RoboDK station: IRB120 3d print.rdk

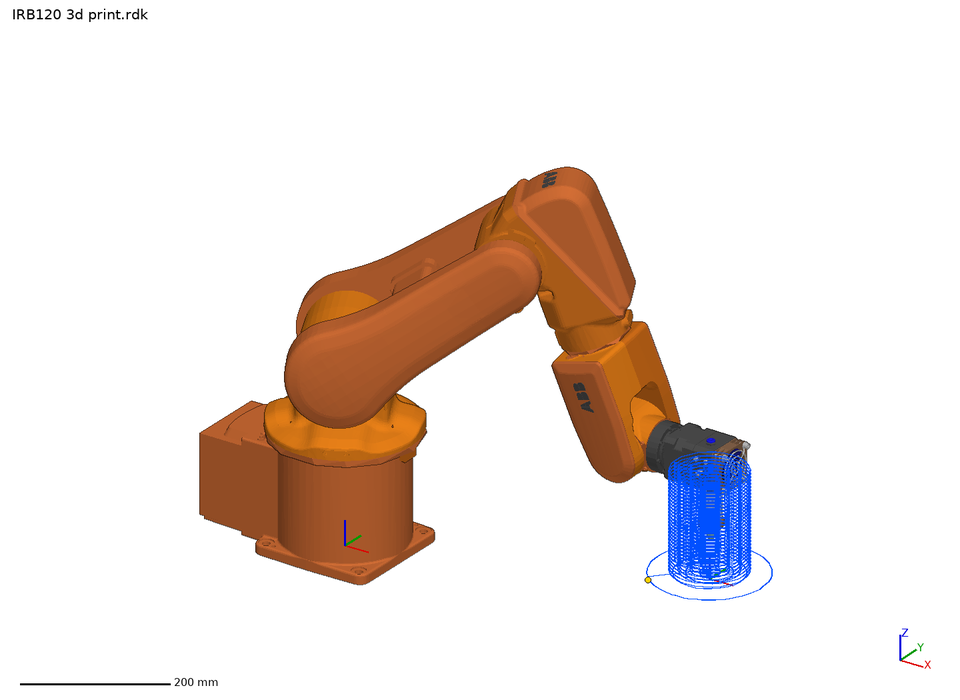
[picture v0: the station drawn from its stored meshes, robots at their saved joint values, targets as dots, program paths as lines]
Station IRB120 3d print (saved by RoboDK 5.2.1). Poses are relative to the parent item; angles as X-Y-Z fixed-axis rotations.
  - frame ABB IRB 120-3/0.6 Base at (0, 0, 0) mm
    - robot ABB IRB 120-3/0.6: 6 axes, payload 3 kg, reach 580 mm, repeatability 0.01 mm, weight 25 kg
        modified DH rows (alpha deg, a mm, theta deg, d mm): 0, 0, 0, 290; -90, 0, -90, 0; 0, 270, 0, 0; -90, 70, 0, 302; 90, 0, 0, 0; -90, 0, 180, 72
        joint limits [-165, -110, -90, -160, -120, -400] to [165, 110, 70, 160, 120, 400]; home [0, 0, 0, 0, 0, 0]; saved at [28.559, 55.09, 16.06, -150.095, 73.514, -189.27]
      - tool Extruder, TCP at (111.33, -10.17, 60.98) mm, rotated rx 0 ry 90 rz 0 deg, size 148.5 x 72.7 x 98.2 mm
  - frame Frame 2 at (454.66, 194.92, 0) mm
    - object Part at (0, 0, 0) mm, size 120 x 120 x 160 mm, geometry from part.sld
  - machining project Print3D settings: C:/Users/Albert/AppData/Local/Temp/Part.stl | rotZ(0) | rotX(0)*rotY(0) | rotZ(0)
  - program Print3D (7572 instructions, listed below)
  - Python program Extruder (listed below)
  - Python program SimulateFinalResult (listed below)
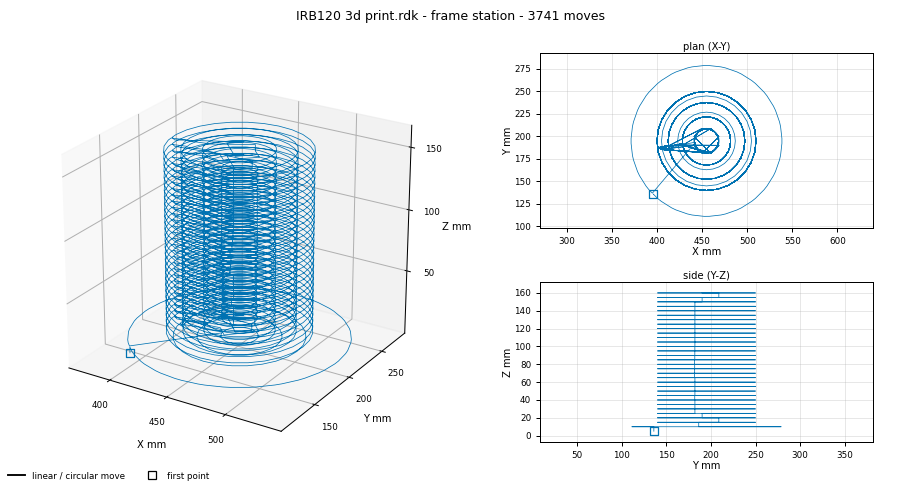
[picture p0: tool path of IRB120 3d print.rdk in frame station, 3741 of 3741 moves have a stored position in this frame; points joined in program order, loops and branches not executed]

--- program Print3D (robot ABB IRB 120-3/0.6) ---
  Set Ref.: Frame 2
  Set Tool: Extruder
  Show Extruder
  Set speed (1000.0 mm/s)
  MoveJ 1 to (-59.03, -59.03, 5) mm, rotated rx 180 ry 0 rz 180 deg; joints [29.08, 61.286, 29.9, -150.915, 91.037, -179.423]
  Set speed (83.3 mm/s)
  MoveL 2 to (-59.03, -59.03, 5) mm, rotated rx 180 ry 0 rz 180 deg; joints [29.08, 61.286, 29.9, -150.915, 91.037, -179.423]
  Call Extruder(-1)
  MoveL 3 to (-59.03, -59.03, 5) mm, rotated rx 180 ry 0 rz 180 deg; joints [29.08, 61.286, 29.9, -150.915, 91.037, -179.423]
  Call Extruder(0.000)
  Set speed (130.0 mm/s)
  MoveL 4 to (-59.03, -59.03, 10) mm, rotated rx 180 ry 0 rz 180 deg; joints [29.08, 60.2, 30.513, -150.918, 90.624, -179.653]
  Call Extruder(-2.000)
  Set speed (40.0 mm/s)
  MoveL 5 to (-59.03, -59.03, 10) mm, rotated rx 180 ry 0 rz 180 deg; joints [29.08, 60.2, 30.513, -150.918, 90.624, -179.653]
  Call Extruder(0.000)
  Set speed (130.0 mm/s)
  MoveL 6 to (-59.03, -59.03, 10) mm, rotated rx 180 ry 0 rz 180 deg; joints [29.08, 60.2, 30.513, -150.918, 90.624, -179.653]
  Call Extruder(2.000)
  Set speed (40.0 mm/s)
  MoveL 7 to (-59.03, -59.03, 10) mm, rotated rx 180 ry 0 rz 180 deg; joints [29.08, 60.2, 30.513, -150.918, 90.624, -179.653]
  Call Extruder(25.861)
  Set speed (30.0 mm/s)
  MoveL 8 to (-54.28, -63.78, 10) mm, rotated rx 180 ry 0 rz 180 deg; joints [27.856, 60.292, 30.1, -152.143, 90.347, -179.817]
  Call Extruder(44.833)
  MoveL 9 to (-50.1, -67.11, 10) mm, rotated rx 180 ry 0 rz -180 deg; joints [26.935, 60.399, 29.628, -153.065, 90.024, -179.988]
  Call Extruder(92.557)
  MoveL 10 to (-38.72, -74.26, 10) mm, rotated rx -180 ry 0 rz -180 deg; joints [24.816, 60.769, 28.068, -155.179, 88.944, -180.488]
  Call Extruder(111.531)
  MoveL 11 to (-33.91, -76.57, 10) mm, rotated rx 180 ry 0 rz 180 deg; joints [24.067, 60.957, 27.309, -155.924, 88.416, -180.708]
  Call Extruder(159.254)
  MoveL 12 to (-21.23, -81.01, 10) mm, rotated rx -180 ry 0 rz -180 deg; joints [22.441, 61.537, 25.081, -157.524, 86.874, -181.292]
  Call Extruder(178.226)
  MoveL 13 to (-16.02, -82.2, 10) mm, rotated rx 180 ry 0 rz 180 deg; joints [21.904, 61.811, 24.081, -158.045, 86.189, -181.535]
  Call Extruder(225.949)
  MoveL 14 to (-2.67, -83.7, 10) mm, rotated rx -180 ry 0 rz -180 deg; joints [20.833, 62.608, 21.313, -159.059, 84.319, -182.169]
  Call Extruder(244.922)
  MoveL 15 to (2.67, -83.7, 10) mm, rotated rx -180 ry 0 rz 180 deg; joints [20.519, 62.966, 20.126, -159.343, 83.532, -182.432]
  Call Extruder(246.414)
  MoveL 16 to (3.09, -83.66, 10) mm, rotated rx 180 ry 0 rz 180 deg; joints [20.502, 62.996, 20.028, -159.358, 83.468, -182.454]
  Call Extruder(292.645)
  MoveL 17 to (16.02, -82.2, 10) mm, rotated rx 180 ry 0 rz 180 deg; joints [19.998, 63.964, 16.96, -159.769, 81.476, -183.127]
  Call Extruder(311.617)
  MoveL 18 to (21.23, -81.01, 10) mm, rotated rx 180 ry 0 rz 180 deg; joints [19.893, 64.397, 15.644, -159.827, 80.641, -183.419]
  Call Extruder(359.340)
  MoveL 19 to (33.91, -76.57, 10) mm, rotated rx -180 ry 0 rz 180 deg; joints [19.872, 65.563, 12.228, -159.706, 78.528, -184.207]
  Call Extruder(378.314)
  MoveL 20 to (38.72, -74.26, 10) mm, rotated rx 180 ry 0 rz -180 deg; joints [19.953, 66.052, 10.842, -159.557, 77.694, -184.542]
  Call Extruder(426.038)
  MoveL 21 to (50.1, -67.11, 10) mm, rotated rx -180 ry 0 rz 180 deg; joints [20.363, 67.333, 7.324, -158.949, 75.638, -185.453]
  Call Extruder(445.010)
  MoveL 22 to (54.28, -63.78, 10) mm, rotated rx -180 ry 0 rz -180 deg; joints [20.601, 67.856, 5.929, -158.621, 74.847, -185.843]
  Call Extruder(492.732)
  MoveL 23 to (63.78, -54.28, 10) mm, rotated rx 180 ry 0 rz -180 deg; joints [21.369, 69.187, 2.461, -157.596, 72.95, -186.892]
  Call Extruder(511.705)
  MoveL 24 to (67.11, -50.1, 10) mm, rotated rx 180 ry 0 rz 180 deg; joints [21.736, 69.715, 1.116, -157.117, 72.241, -187.336]
  Call Extruder(559.428)
  MoveL 25 to (74.26, -38.72, 10) mm, rotated rx -180 ry 0 rz -180 deg; joints [22.792, 71.021, -2.147, -155.749, 70.593, -188.513]
  Call Extruder(578.402)
  MoveL 26 to (76.57, -33.91, 10) mm, rotated rx 180 ry 0 rz -180 deg; joints [23.26, 71.524, -3.38, -155.15, 70, -189.001]
  Call Extruder(626.125)
  MoveL 27 to (81.01, -21.23, 10) mm, rotated rx 180 ry 0 rz 180 deg; joints [24.541, 72.722, -6.277, -153.522, 68.682, -190.264]
  Call Extruder(645.097)
  MoveL 28 to (82.2, -16.02, 10) mm, rotated rx -180 ry 0 rz -180 deg; joints [25.087, 73.164, -7.333, -152.836, 68.235, -190.773]
  Call Extruder(692.820)
  MoveL 29 to (83.7, -2.67, 10) mm, rotated rx 180 ry 0 rz -180 deg; joints [26.535, 74.169, -9.705, -151.04, 67.315, -192.048]
  Call Extruder(711.794)
  MoveL 30 to (83.7, 2.67, 10) mm, rotated rx 180 ry 0 rz -180 deg; joints [27.136, 74.518, -10.521, -150.306, 67.036, -192.543]
  Call Extruder(759.517)
  MoveL 31 to (82.2, 16.02, 10) mm, rotated rx 180 ry 0 rz 180 deg; joints [28.7, 75.248, -12.216, -148.438, 66.561, -193.731]
  Call Extruder(778.488)
  MoveL 32 to (81.01, 21.23, 10) mm, rotated rx 180 ry 0 rz -180 deg; joints [29.338, 75.474, -12.736, -147.696, 66.465, -194.17]
  Call Extruder(826.211)
  MoveL 33 to (76.57, 33.91, 10) mm, rotated rx 180 ry 0 rz -180 deg; joints [30.97, 75.863, -13.631, -145.853, 66.455, -195.16]
  Call Extruder(845.186)
  MoveL 34 to (74.26, 38.72, 10) mm, rotated rx 180 ry 0 rz 180 deg; joints [31.625, 75.944, -13.816, -145.138, 66.542, -195.499]
  Call Extruder(892.909)
  MoveL 35 to (67.11, 50.1, 10) mm, rotated rx 180 ry 0 rz 180 deg; joints [33.281, 75.955, -13.842, -143.401, 66.982, -196.192]
  Call Extruder(911.881)
  MoveL 36 to (63.78, 54.28, 10) mm, rotated rx 180 ry 0 rz 180 deg; joints [33.937, 75.884, -13.678, -142.741, 67.241, -196.398]
  Call Extruder(959.604)
  MoveL 37 to (54.28, 63.78, 10) mm, rotated rx 180 ry 0 rz 180 deg; joints [35.572, 75.515, -12.832, -141.168, 68.083, -196.723]
  Call Extruder(978.576)
  MoveL 38 to (50.1, 67.11, 10) mm, rotated rx 180 ry 0 rz 180 deg; joints [36.21, 75.298, -12.331, -140.581, 68.487, -196.774]
  Call Extruder(1026.299)
  MoveL 39 to (38.72, 74.26, 10) mm, rotated rx -180 ry 0 rz 180 deg; joints [37.78, 74.586, -10.68, -139.203, 69.657, -196.701]
  Call Extruder(1045.274)
  MoveL 40 to (33.91, 76.57, 10) mm, rotated rx -180 ry 0 rz 180 deg; joints [38.384, 74.244, -9.88, -138.697, 70.175, -196.593]
  Call Extruder(1092.996)
  MoveL 41 to (21.23, 81.01, 10) mm, rotated rx 180 ry 0 rz -180 deg; joints [39.84, 73.253, -7.544, -137.529, 71.587, -196.127]
  Call Extruder(1111.968)
  MoveL 42 to (16.02, 82.2, 10) mm, rotated rx 180 ry 0 rz 180 deg; joints [40.39, 72.815, -6.501, -137.108, 72.183, -195.868]
  Call Extruder(1159.691)
  MoveL 43 to (2.67, 83.7, 10) mm, rotated rx 180 ry 0 rz -180 deg; joints [41.682, 71.626, -3.63, -136.158, 73.751, -195.042]
  Call Extruder(1178.665)
  MoveL 44 to (-2.67, 83.7, 10) mm, rotated rx 180 ry 0 rz -180 deg; joints [42.155, 71.126, -2.405, -135.827, 74.393, -194.649]
  Call Extruder(1226.388)
  MoveL 45 to (-16.02, 82.2, 10) mm, rotated rx 180 ry 0 rz -180 deg; joints [43.227, 69.824, 0.84, -135.111, 76.039, -193.513]
  Call Extruder(1245.360)
  MoveL 46 to (-21.23, 81.01, 10) mm, rotated rx 180 ry 0 rz -180 deg; joints [43.6, 69.297, 2.181, -134.877, 76.7, -193.009]
  Call Extruder(1293.082)
  MoveL 47 to (-33.91, 76.57, 10) mm, rotated rx -180 ry 0 rz -180 deg; joints [44.387, 67.965, 5.64, -134.424, 78.363, -191.629]
  Call Extruder(1312.057)
  MoveL 48 to (-38.72, 74.26, 10) mm, rotated rx 180 ry 0 rz -180 deg; joints [44.633, 67.441, 7.035, -134.302, 79.021, -191.043]
  Call Extruder(1359.780)
  MoveL 49 to (-50.1, 67.11, 10) mm, rotated rx 180 ry 0 rz 180 deg; joints [45.066, 66.155, 10.554, -134.156, 80.655, -189.494]
  Call Extruder(1378.752)
  MoveL 50 to (-54.28, 63.78, 10) mm, rotated rx -180 ry 0 rz -180 deg; joints [45.158, 65.663, 11.942, -134.167, 81.294, -188.857]
  Call Extruder(1380.244)
  MoveL 51 to (-54.57, 63.48, 10) mm, rotated rx 180 ry 0 rz 180 deg; joints [45.158, 65.625, 12.051, -134.174, 81.343, -188.806]
  Call Extruder(1426.475)
  MoveL 52 to (-63.78, 54.28, 10) mm, rotated rx 180 ry 0 rz 180 deg; joints [45.163, 64.489, 15.368, -134.385, 82.867, -187.23]
  Call Extruder(1445.447)
  MoveL 53 to (-67.11, 50.1, 10) mm, rotated rx 180 ry 0 rz -180 deg; joints [45.071, 64.052, 16.69, -134.554, 83.476, -186.583]
  Call Extruder(1493.170)
  MoveL 54 to (-74.26, 38.72, 10) mm, rotated rx 180 ry 0 rz -180 deg; joints [44.58, 63.043, 19.875, -135.2, 84.962, -184.984]
  Call Extruder(1512.145)
  MoveL 55 to (-76.57, 33.91, 10) mm, rotated rx 180 ry 0 rz 180 deg; joints [44.279, 62.68, 21.071, -135.55, 85.53, -184.372]
  Call Extruder(1559.868)
  MoveL 56 to (-81.01, 21.23, 10) mm, rotated rx -180 ry 0 rz 180 deg; joints [43.242, 61.871, 23.866, -136.679, 86.896, -182.923]
  Call Extruder(1578.839)
  MoveL 57 to (-82.2, 16.02, 10) mm, rotated rx 180 ry 0 rz 180 deg; joints [42.718, 61.592, 24.879, -137.228, 87.408, -182.396]
  Call Extruder(1626.562)
  MoveL 58 to (-83.7, 2.67, 10) mm, rotated rx 180 ry 0 rz -180 deg; joints [41.124, 60.999, 27.142, -138.861, 88.6, -181.223]
  Call Extruder(1645.536)
  MoveL 59 to (-83.7, -2.67, 10) mm, rotated rx 180 ry 0 rz 180 deg; joints [40.386, 60.806, 27.917, -139.607, 89.027, -180.828]
  Call Extruder(1693.259)
  MoveL 60 to (-82.2, -16.02, 10) mm, rotated rx -180 ry 0 rz 180 deg; joints [38.292, 60.424, 29.52, -141.708, 89.956, -180.035]
  Call Extruder(1712.231)
  MoveL 61 to (-81.01, -21.23, 10) mm, rotated rx 180 ry 0 rz 180 deg; joints [37.38, 60.313, 30.01, -142.62, 90.256, -179.804]
  Call Extruder(1759.954)
  MoveL 62 to (-76.57, -33.91, 10) mm, rotated rx 180 ry 0 rz -180 deg; joints [34.932, 60.126, 30.851, -145.065, 90.802, -179.44]
  Call Extruder(1778.928)
  MoveL 63 to (-74.26, -38.72, 10) mm, rotated rx 180 ry 0 rz 180 deg; joints [33.918, 60.089, 31.025, -146.077, 90.924, -179.378]
  Call Extruder(1826.651)
  MoveL 64 to (-67.11, -50.1, 10) mm, rotated rx -180 ry 0 rz 180 deg; joints [31.335, 60.084, 31.049, -148.66, 90.968, -179.411]
  Call Extruder(1845.623)
  MoveL 65 to (-63.78, -54.28, 10) mm, rotated rx -180 ry 0 rz 180 deg; joints [30.319, 60.117, 30.895, -149.677, 90.873, -179.489]
  Call Extruder(1864.157)
  MoveL 66 to (-60.09, -57.97, 10) mm, rotated rx -180 ry 0 rz 180 deg; joints [29.356, 60.181, 30.601, -150.642, 90.682, -179.617]
  Call Extruder(1862.157)
  Set speed (40.0 mm/s)
  MoveL 67 to (-60.09, -57.97, 10) mm, rotated rx -180 ry 0 rz 180 deg; joints [29.356, 60.181, 30.601, -150.642, 90.682, -179.617]
  Call Extruder(0.000)
  Set speed (130.0 mm/s)
  MoveL 68 to (-13.65, -3.12, 10) mm, rotated rx 180 ry 0 rz 180 deg; joints [33.254, 64.706, 14.722, -146.295, 81.174, -185.844]
  Call Extruder(2.000)
  Set speed (40.0 mm/s)
  MoveL 69 to (-13.65, -3.12, 10) mm, rotated rx 180 ry 0 rz 180 deg; joints [33.254, 64.706, 14.722, -146.295, 81.174, -185.844]
  Call Extruder(13.137)
  Set speed (30.0 mm/s)
  MoveL 70 to (-12.62, -6.08, 10) mm, rotated rx 180 ry 0 rz -180 deg; joints [32.78, 64.642, 14.909, -146.783, 81.23, -185.702]
  Call Extruder(24.274)
  MoveL 71 to (-10.95, -8.73, 10) mm, rotated rx 180 ry 0 rz 180 deg; joints [32.291, 64.641, 14.914, -147.275, 81.185, -185.624]
  Call Extruder(35.413)
  MoveL 72 to (-8.73, -10.95, 10) mm, rotated rx 180 ry 0 rz 180 deg; joints [31.815, 64.7, 14.737, -147.745, 81.039, -185.614]
  Call Extruder(46.550)
  MoveL 73 to (-6.08, -12.62, 10) mm, rotated rx -180 ry 0 rz -180 deg; joints [31.379, 64.819, 14.387, -148.165, 80.799, -185.669]
  Call Extruder(57.687)
  MoveL 74 to (-3.12, -13.65, 10) mm, rotated rx 180 ry 0 rz 180 deg; joints [31.005, 64.991, 13.881, -148.513, 80.478, -185.786]
  Call Extruder(68.825)
  MoveL 75 to (0, -14, 10) mm, rotated rx -180 ry 0 rz -180 deg; joints [30.713, 65.21, 13.244, -148.77, 80.091, -185.957]
  Call Extruder(79.963)
  MoveL 76 to (3.12, -13.65, 10) mm, rotated rx 180 ry 0 rz -180 deg; joints [30.517, 65.465, 12.508, -148.924, 79.659, -186.174]
  Call Extruder(91.100)
  MoveL 77 to (6.08, -12.62, 10) mm, rotated rx 180 ry 0 rz -180 deg; joints [30.425, 65.744, 11.711, -148.967, 79.205, -186.429]
  Call Extruder(102.237)
  MoveL 78 to (8.73, -10.95, 10) mm, rotated rx -180 ry 0 rz -180 deg; joints [30.439, 66.034, 10.892, -148.9, 78.754, -186.71]
  Call Extruder(113.376)
  MoveL 79 to (10.95, -8.73, 10) mm, rotated rx 180 ry 0 rz -180 deg; joints [30.556, 66.321, 10.092, -148.727, 78.328, -187.005]
  Call Extruder(124.513)
  MoveL 80 to (12.62, -6.08, 10) mm, rotated rx 180 ry 0 rz -180 deg; joints [30.767, 66.589, 9.35, -148.461, 77.95, -187.301]
  Call Extruder(135.650)
  MoveL 81 to (13.65, -3.12, 10) mm, rotated rx 180 ry 0 rz 180 deg; joints [31.062, 66.824, 8.705, -148.115, 77.64, -187.585]
  Call Extruder(146.788)
  MoveL 82 to (14, 0, 10) mm, rotated rx 180 ry 0 rz 180 deg; joints [31.425, 67.014, 8.189, -147.709, 77.412, -187.842]
  Call Extruder(157.926)
  MoveL 83 to (13.65, 3.12, 10) mm, rotated rx 180 ry 0 rz 180 deg; joints [31.837, 67.147, 7.827, -147.263, 77.276, -188.06]
  Call Extruder(169.063)
  MoveL 84 to (12.62, 6.08, 10) mm, rotated rx 180 ry 0 rz 180 deg; joints [32.281, 67.217, 7.639, -146.798, 77.239, -188.225]
  Call Extruder(180.200)
  MoveL 85 to (10.95, 8.73, 10) mm, rotated rx -180 ry 0 rz -180 deg; joints [32.735, 67.219, 7.634, -146.337, 77.302, -188.328]
  Call Extruder(191.339)
  MoveL 86 to (8.73, 10.95, 10) mm, rotated rx -180 ry 0 rz 180 deg; joints [33.18, 67.153, 7.811, -145.9, 77.46, -188.363]
  Call Extruder(202.476)
  MoveL 87 to (6.08, 12.62, 10) mm, rotated rx 180 ry 0 rz -180 deg; joints [33.595, 67.023, 8.163, -145.507, 77.703, -188.325]
  Call Extruder(213.613)
  MoveL 88 to (3.12, 13.65, 10) mm, rotated rx -180 ry 0 rz 180 deg; joints [33.96, 66.837, 8.671, -145.176, 78.02, -188.216]
  Call Extruder(224.751)
  MoveL 89 to (0, 14, 10) mm, rotated rx -180 ry 0 rz 180 deg; joints [34.26, 66.604, 9.309, -144.922, 78.395, -188.041]
  Call Extruder(235.889)
  MoveL 90 to (-3.12, 13.65, 10) mm, rotated rx 180 ry 0 rz -180 deg; joints [34.477, 66.337, 10.046, -144.757, 78.809, -187.808]
  Call Extruder(247.026)
  MoveL 91 to (-6.08, 12.62, 10) mm, rotated rx 180 ry 0 rz 180 deg; joints [34.599, 66.051, 10.844, -144.691, 79.244, -187.53]
  Call Extruder(258.163)
  MoveL 92 to (-8.73, 10.95, 10) mm, rotated rx -180 ry 0 rz -180 deg; joints [34.62, 65.761, 11.663, -144.727, 79.678, -187.223]
  Call Extruder(269.302)
  MoveL 93 to (-10.95, 8.73, 10) mm, rotated rx 180 ry 0 rz -180 deg; joints [34.534, 65.481, 12.463, -144.867, 80.092, -186.904]
  Call Extruder(280.439)
  MoveL 94 to (-12.62, 6.08, 10) mm, rotated rx 180 ry 0 rz -180 deg; joints [34.344, 65.224, 13.203, -145.106, 80.465, -186.59]
  Call Extruder(291.576)
  MoveL 95 to (-13.65, 3.12, 10) mm, rotated rx 180 ry 0 rz 180 deg; joints [34.057, 65.003, 13.846, -145.434, 80.78, -186.299]
  Call Extruder(302.714)
  MoveL 96 to (-14, 0, 10) mm, rotated rx 180 ry 0 rz 180 deg; joints [33.688, 64.828, 14.361, -145.837, 81.021, -186.046]
  Call Extruder(308.524)
  MoveL 97 to (-13.82, -1.63, 10) mm, rotated rx 180 ry 0 rz 180 deg; joints [33.462, 64.764, 14.55, -146.075, 81.101, -185.94]
  Set speed (130.0 mm/s)
  MoveL 98 to (-31.39, -5.11, 10) mm, rotated rx 180 ry 0 rz -180 deg; joints [34.564, 63.427, 18.638, -145.178, 83.473, -184.521]
  Call Extruder(315.669)
  Set speed (30.0 mm/s)
  MoveL 99 to (-31.17, -7.11, 10) mm, rotated rx -180 ry 0 rz -180 deg; joints [34.275, 63.356, 18.867, -145.478, 83.579, -184.398]
  Call Extruder(341.097)
  MoveL 100 to (-28.8, -13.87, 10) mm, rotated rx 180 ry 0 rz -180 deg; joints [33.142, 63.221, 19.297, -146.634, 83.741, -184.107]
  Call Extruder(366.525)
  MoveL 101 to (-25, -19.93, 10) mm, rotated rx 180 ry 0 rz 180 deg; joints [31.969, 63.217, 19.31, -147.811, 83.665, -183.973]
  Call Extruder(391.953)
  MoveL 102 to (-19.93, -24.99, 10) mm, rotated rx 180 ry 0 rz -180 deg; joints [30.832, 63.344, 18.904, -148.936, 83.349, -183.991]
  Call Extruder(417.381)
  MoveL 103 to (-13.87, -28.8, 10) mm, rotated rx 180 ry 0 rz 180 deg; joints [29.802, 63.598, 18.1, -149.937, 82.802, -184.148]
  Call Extruder(442.809)
  MoveL 104 to (-7.11, -31.17, 10) mm, rotated rx 180 ry 0 rz -180 deg; joints [28.939, 63.971, 16.94, -150.753, 82.054, -184.426]
  Call Extruder(468.237)
  MoveL 105 to (0, -31.97, 10) mm, rotated rx -180 ry 0 rz 180 deg; joints [28.289, 64.45, 15.484, -151.338, 81.147, -184.809]
  Call Extruder(493.666)
  MoveL 106 to (7.11, -31.17, 10) mm, rotated rx 180 ry 0 rz -180 deg; joints [27.879, 65.017, 13.804, -151.665, 80.133, -185.279]
  Call Extruder(519.094)
  MoveL 107 to (13.87, -28.8, 10) mm, rotated rx -180 ry 0 rz -180 deg; joints [27.717, 65.648, 11.985, -151.726, 79.07, -185.823]
  Call Extruder(544.522)
  MoveL 108 to (19.93, -24.99, 10) mm, rotated rx 180 ry 0 rz -180 deg; joints [27.799, 66.313, 10.114, -151.526, 78.018, -186.424]
  Call Extruder(569.950)
  MoveL 109 to (24.99, -19.93, 10) mm, rotated rx 180 ry 0 rz 180 deg; joints [28.108, 66.978, 8.284, -151.089, 77.033, -187.064]
  Call Extruder(595.378)
  MoveL 110 to (28.8, -13.87, 10) mm, rotated rx 180 ry 0 rz 180 deg; joints [28.617, 67.609, 6.586, -150.445, 76.167, -187.721]
  Call Extruder(620.806)
  MoveL 111 to (31.17, -7.11, 10) mm, rotated rx 180 ry 0 rz 180 deg; joints [29.297, 68.168, 5.106, -149.634, 75.464, -188.366]
  Call Extruder(646.234)
  MoveL 112 to (31.97, 0, 10) mm, rotated rx 180 ry 0 rz -180 deg; joints [30.112, 68.623, 3.917, -148.702, 74.957, -188.967]
  Call Extruder(671.663)
  MoveL 113 to (31.17, 7.11, 10) mm, rotated rx 180 ry 0 rz 180 deg; joints [31.024, 68.945, 3.083, -147.696, 74.668, -189.491]
  Call Extruder(697.091)
  MoveL 114 to (28.8, 13.87, 10) mm, rotated rx 180 ry 0 rz 180 deg; joints [31.996, 69.114, 2.648, -146.663, 74.608, -189.904]
  Call Extruder(722.519)
  MoveL 115 to (24.99, 19.93, 10) mm, rotated rx 180 ry 0 rz -180 deg; joints [32.988, 69.119, 2.636, -145.648, 74.775, -190.175]
  Call Extruder(747.947)
  MoveL 116 to (19.93, 25, 10) mm, rotated rx 180 ry 0 rz -180 deg; joints [33.962, 68.96, 3.046, -144.694, 75.154, -190.285]
  Call Extruder(773.375)
  MoveL 117 to (13.87, 28.8, 10) mm, rotated rx 180 ry 0 rz 180 deg; joints [34.879, 68.646, 3.858, -143.837, 75.721, -190.219]
  Call Extruder(798.803)
  MoveL 118 to (7.11, 31.17, 10) mm, rotated rx 180 ry 0 rz -180 deg; joints [35.701, 68.198, 5.027, -143.111, 76.445, -189.977]
  Call Extruder(824.231)
  MoveL 119 to (0, 31.97, 10) mm, rotated rx -180 ry 0 rz -180 deg; joints [36.389, 67.644, 6.493, -142.542, 77.288, -189.569]
  Call Extruder(849.660)
  MoveL 120 to (-7.11, 31.17, 10) mm, rotated rx 180 ry 0 rz -180 deg; joints [36.91, 67.017, 8.18, -142.157, 78.212, -189.018]
  Call Extruder(875.088)
  MoveL 121 to (-13.87, 28.8, 10) mm, rotated rx 180 ry 0 rz -180 deg; joints [37.231, 66.352, 10.004, -141.976, 79.175, -188.355]
  Call Extruder(900.516)
  MoveL 122 to (-19.93, 25, 10) mm, rotated rx 180 ry 0 rz -180 deg; joints [37.327, 65.686, 11.875, -142.015, 80.138, -187.618]
  Call Extruder(925.944)
  MoveL 123 to (-25, 19.93, 10) mm, rotated rx 180 ry 0 rz -180 deg; joints [37.18, 65.053, 13.7, -142.284, 81.06, -186.852]
  Call Extruder(951.372)
  MoveL 124 to (-28.8, 13.87, 10) mm, rotated rx -180 ry 0 rz 180 deg; joints [36.784, 64.481, 15.391, -142.784, 81.904, -186.105]
  Call Extruder(976.800)
  MoveL 125 to (-31.17, 7.11, 10) mm, rotated rx -180 ry 0 rz 180 deg; joints [36.147, 63.996, 16.862, -143.503, 82.629, -185.422]
  Call Extruder(1002.229)
  MoveL 126 to (-31.97, 0, 10) mm, rotated rx -180 ry 0 rz -180 deg; joints [35.297, 63.617, 18.041, -144.416, 83.199, -184.843]
  Call Extruder(1015.184)
  MoveL 127 to (-31.56, -3.62, 10) mm, rotated rx 180 ry 0 rz 180 deg; joints [34.778, 63.482, 18.466, -144.955, 83.393, -184.614]
  Set speed (130.0 mm/s)
  MoveL 128 to (-49.14, -7.11, 10) mm, rotated rx 180 ry 0 rz 180 deg; joints [35.996, 62.3, 22.36, -143.885, 85.682, -183.144]
  Call Extruder(1029.474)
  Set speed (30.0 mm/s)
  MoveL 129 to (-48.69, -11.11, 10) mm, rotated rx -180 ry 0 rz 180 deg; joints [35.397, 62.167, 22.819, -144.499, 85.915, -182.909]
  Call Extruder(1069.192)
  MoveL 130 to (-44.99, -21.67, 10) mm, rotated rx 180 ry 0 rz 180 deg; joints [33.543, 61.974, 23.498, -146.375, 86.227, -182.506]
  Call Extruder(1108.911)
  MoveL 131 to (-39.04, -31.13, 10) mm, rotated rx 180 ry 0 rz -180 deg; joints [31.612, 61.969, 23.517, -148.308, 86.157, -182.37]
  Call Extruder(1148.630)
  MoveL 132 to (-31.13, -39.04, 10) mm, rotated rx 180 ry 0 rz 180 deg; joints [29.75, 62.151, 22.876, -150.157, 85.684, -182.472]
  Call Extruder(1188.349)
  MoveL 133 to (-21.67, -44.99, 10) mm, rotated rx 180 ry 0 rz 180 deg; joints [28.087, 62.519, 21.611, -151.787, 84.823, -182.771]
  Call Extruder(1228.067)
  MoveL 134 to (-11.11, -48.68, 10) mm, rotated rx 180 ry 0 rz 180 deg; joints [26.732, 63.069, 19.789, -153.089, 83.625, -183.226]
  Call Extruder(1267.786)
  MoveL 135 to (0, -49.94, 10) mm, rotated rx -180 ry 0 rz 180 deg; joints [25.75, 63.788, 17.507, -153.989, 82.165, -183.806]
  Call Extruder(1307.505)
  MoveL 136 to (11.11, -48.68, 10) mm, rotated rx 180 ry 0 rz -180 deg; joints [25.174, 64.652, 14.88, -154.454, 80.536, -184.494]
  Call Extruder(1347.223)
  MoveL 137 to (21.67, -44.99, 10) mm, rotated rx -180 ry 0 rz -180 deg; joints [25, 65.63, 12.037, -154.483, 78.838, -185.279]
  Call Extruder(1386.942)
  MoveL 138 to (31.13, -39.04, 10) mm, rotated rx 180 ry 0 rz 180 deg; joints [25.205, 66.675, 9.114, -154.103, 77.166, -186.155]
  Call Extruder(1426.661)
  MoveL 139 to (39.04, -31.13, 10) mm, rotated rx 180 ry 0 rz 180 deg; joints [25.746, 67.735, 6.25, -153.355, 75.611, -187.107]
  Call Extruder(1466.380)
  MoveL 140 to (44.99, -21.67, 10) mm, rotated rx 180 ry 0 rz 180 deg; joints [26.577, 68.751, 3.584, -152.3, 74.253, -188.109]
  Call Extruder(1506.098)
  MoveL 141 to (48.69, -11.11, 10) mm, rotated rx 180 ry 0 rz 180 deg; joints [27.644, 69.663, 1.248, -151.003, 73.16, -189.122]
  Call Extruder(1545.817)
  MoveL 142 to (49.94, 0, 10) mm, rotated rx 180 ry 0 rz 180 deg; joints [28.895, 70.412, -0.634, -149.537, 72.384, -190.093]
  Call Extruder(1585.536)
  MoveL 143 to (48.68, 11.11, 10) mm, rotated rx 180 ry 0 rz 180 deg; joints [30.275, 70.946, -1.96, -147.979, 71.959, -190.961]
  Call Extruder(1625.254)
  MoveL 144 to (44.99, 21.67, 10) mm, rotated rx -180 ry 0 rz -180 deg; joints [31.735, 71.227, -2.653, -146.402, 71.9, -191.662]
  Call Extruder(1664.973)
  MoveL 145 to (39.04, 31.14, 10) mm, rotated rx 180 ry 0 rz -180 deg; joints [33.221, 71.235, -2.673, -144.871, 72.196, -192.141]
  Call Extruder(1704.692)
  MoveL 146 to (31.13, 39.04, 10) mm, rotated rx 180 ry 0 rz -180 deg; joints [34.683, 70.969, -2.019, -143.445, 72.821, -192.352]
  Call Extruder(1744.411)
  MoveL 147 to (21.67, 44.99, 10) mm, rotated rx -180 ry 0 rz -180 deg; joints [36.069, 70.449, -0.728, -142.17, 73.731, -192.273]
  Call Extruder(1784.129)
  MoveL 148 to (11.11, 48.69, 10) mm, rotated rx 180 ry 0 rz -180 deg; joints [37.329, 69.712, 1.124, -141.085, 74.869, -191.9]
  Call Extruder(1823.848)
  MoveL 149 to (0, 49.94, 10) mm, rotated rx 180 ry 0 rz 180 deg; joints [38.408, 68.809, 3.436, -140.223, 76.174, -191.251]
  Call Extruder(1863.567)
  MoveL 150 to (-11.11, 48.68, 10) mm, rotated rx -180 ry 0 rz -180 deg; joints [39.255, 67.797, 6.086, -139.616, 77.587, -190.362]
  Call Extruder(1903.286)
  MoveL 151 to (-21.67, 44.99, 10) mm, rotated rx 180 ry 0 rz 180 deg; joints [39.815, 66.737, 8.942, -139.293, 79.048, -189.283]
  Call Extruder(1943.005)
  MoveL 152 to (-31.14, 39.04, 10) mm, rotated rx 180 ry 0 rz 180 deg; joints [40.04, 65.69, 11.866, -139.288, 80.504, -188.08]
  Call Extruder(1982.723)
  MoveL 153 to (-39.04, 31.14, 10) mm, rotated rx -180 ry 0 rz 180 deg; joints [39.89, 64.707, 14.717, -139.627, 81.905, -186.828]
  Call Extruder(2022.442)
  MoveL 154 to (-44.99, 21.67, 10) mm, rotated rx 180 ry 0 rz -180 deg; joints [39.337, 63.835, 17.36, -140.329, 83.201, -185.608]
  Call Extruder(2062.161)
  MoveL 155 to (-48.68, 11.11, 10) mm, rotated rx 180 ry 0 rz 180 deg; joints [38.379, 63.107, 19.666, -141.398, 84.341, -184.502]
  Call Extruder(2101.879)
  MoveL 156 to (-49.94, 0, 10) mm, rotated rx 180 ry 0 rz -180 deg; joints [37.044, 62.547, 21.518, -142.808, 85.266, -183.584]
  Call Extruder(2121.981)
  MoveL 157 to (-49.3, -5.62, 10) mm, rotated rx -180 ry 0 rz -180 deg; joints [36.217, 62.35, 22.187, -143.658, 85.595, -183.234]
  Set speed (130.0 mm/s)
  MoveL 158 to (-45.45, -8.72, 10) mm, rotated rx 180 ry 0 rz -180 deg; joints [35.41, 62.44, 21.879, -144.457, 85.373, -183.299]
  MoveL 159 to (-45.45, -8.72, 15) mm, rotated rx 180 ry 0 rz -180 deg; joints [35.41, 61.424, 22.455, -144.436, 85.014, -183.556]
  MoveL 160 to (-26.25, -4.54, 15) mm, rotated rx -180 ry 0 rz 180 deg; joints [34.172, 62.794, 18.095, -145.489, 82.472, -185.147]
  Call Extruder(2124.213)
  Set speed (60.0 mm/s)
  MoveL 161 to (-26.09, -5.96, 15) mm, rotated rx 180 ry 0 rz -180 deg; joints [33.969, 62.741, 18.258, -145.701, 82.545, -185.058]
  Call Extruder(2133.578)
  MoveL 162 to (-24.12, -11.61, 15) mm, rotated rx 180 ry 0 rz 180 deg; joints [33.033, 62.624, 18.618, -146.659, 82.666, -184.801]
  Call Extruder(2142.943)
  MoveL 163 to (-20.93, -16.69, 15) mm, rotated rx 180 ry 0 rz 180 deg; joints [32.066, 62.621, 18.628, -147.632, 82.592, -184.672]
  Call Extruder(2152.308)
  MoveL 164 to (-16.69, -20.93, 15) mm, rotated rx -180 ry 0 rz -180 deg; joints [31.126, 62.731, 18.288, -148.56, 82.321, -184.67]
  Call Extruder(2161.673)
  MoveL 165 to (-11.61, -24.11, 15) mm, rotated rx 180 ry 0 rz -180 deg; joints [30.272, 62.952, 17.616, -149.388, 81.863, -184.787]
  Call Extruder(2171.038)
  MoveL 166 to (-5.96, -26.09, 15) mm, rotated rx -180 ry 0 rz -180 deg; joints [29.552, 63.275, 16.646, -150.064, 81.243, -185.01]
  Call Extruder(2180.403)
  MoveL 167 to (0, -26.77, 15) mm, rotated rx 180 ry 0 rz 180 deg; joints [29.003, 63.688, 15.427, -150.554, 80.493, -185.327]
  Call Extruder(2189.768)
  MoveL 168 to (5.96, -26.09, 15) mm, rotated rx -180 ry 0 rz 180 deg; joints [28.65, 64.174, 14.02, -150.832, 79.657, -185.723]
  Call Extruder(2199.133)
  MoveL 169 to (11.61, -24.11, 15) mm, rotated rx 180 ry 0 rz 180 deg; joints [28.503, 64.711, 12.497, -150.889, 78.78, -186.184]
  Call Extruder(2208.498)
  MoveL 170 to (16.69, -20.93, 15) mm, rotated rx 180 ry 0 rz -180 deg; joints [28.559, 65.275, 10.931, -150.731, 77.912, -186.694]
  Call Extruder(2217.863)
  MoveL 171 to (20.93, -16.69, 15) mm, rotated rx 180 ry 0 rz 180 deg; joints [28.808, 65.836, 9.401, -150.373, 77.098, -187.237]
  Call Extruder(2227.228)
  MoveL 172 to (24.12, -11.61, 15) mm, rotated rx 180 ry 0 rz 180 deg; joints [29.229, 66.365, 7.982, -149.84, 76.381, -187.791]
  Call Extruder(2236.593)
  MoveL 173 to (26.09, -5.96, 15) mm, rotated rx 180 ry 0 rz -180 deg; joints [29.796, 66.832, 6.746, -149.164, 75.799, -188.332]
  Call Extruder(2245.958)
  MoveL 174 to (26.77, 0, 15) mm, rotated rx -180 ry 0 rz -180 deg; joints [30.482, 67.211, 5.755, -148.383, 75.378, -188.834]
  Call Extruder(2255.323)
  MoveL 175 to (26.09, 5.96, 15) mm, rotated rx -180 ry 0 rz 180 deg; joints [31.252, 67.479, 5.061, -147.536, 75.137, -189.268]
  Call Extruder(2264.688)
  MoveL 176 to (24.11, 11.61, 15) mm, rotated rx -180 ry 0 rz -180 deg; joints [32.076, 67.619, 4.699, -146.664, 75.086, -189.609]
  Call Extruder(2274.053)
  MoveL 177 to (20.93, 16.69, 15) mm, rotated rx 180 ry 0 rz -180 deg; joints [32.917, 67.623, 4.688, -145.805, 75.223, -189.832]
  Call Extruder(2283.418)
  MoveL 178 to (16.69, 20.93, 15) mm, rotated rx 180 ry 0 rz -180 deg; joints [33.742, 67.491, 5.03, -144.996, 75.537, -189.921]
  Call Extruder(2292.783)
  MoveL 179 to (11.61, 24.12, 15) mm, rotated rx -180 ry 0 rz -180 deg; joints [34.517, 67.23, 5.706, -144.269, 76.008, -189.867]
  Call Extruder(2302.148)
  MoveL 180 to (5.96, 26.09, 15) mm, rotated rx 180 ry 0 rz -180 deg; joints [35.208, 66.857, 6.681, -143.654, 76.612, -189.669]
  Call Extruder(2311.513)
  MoveL 181 to (0, 26.77, 15) mm, rotated rx 180 ry 0 rz 180 deg; joints [35.784, 66.394, 7.904, -143.176, 77.318, -189.335]
  Call Extruder(2320.878)
  MoveL 182 to (-5.96, 26.09, 15) mm, rotated rx 180 ry 0 rz 180 deg; joints [36.214, 65.868, 9.314, -142.858, 78.092, -188.883]
  Call Extruder(2330.243)
  MoveL 183 to (-11.61, 24.12, 15) mm, rotated rx 180 ry 0 rz 180 deg; joints [36.473, 65.308, 10.839, -142.715, 78.9, -188.34]
  Call Extruder(2339.608)
  MoveL 184 to (-16.69, 20.93, 15) mm, rotated rx 180 ry 0 rz 180 deg; joints [36.542, 64.744, 12.405, -142.761, 79.706, -187.735]
  Call Extruder(2348.973)
  MoveL 185 to (-20.93, 16.69, 15) mm, rotated rx 180 ry 0 rz -180 deg; joints [36.407, 64.204, 13.933, -143.001, 80.477, -187.106]
  Call Extruder(2358.338)
  MoveL 186 to (-24.12, 11.61, 15) mm, rotated rx 180 ry 0 rz 180 deg; joints [36.065, 63.715, 15.349, -143.433, 81.178, -186.49]
  Call Extruder(2367.702)
  MoveL 187 to (-26.09, 5.96, 15) mm, rotated rx -180 ry 0 rz 180 deg; joints [35.528, 63.297, 16.58, -144.046, 81.776, -185.923]
  Call Extruder(2377.068)
  MoveL 188 to (-26.77, 0, 15) mm, rotated rx 180 ry 0 rz 180 deg; joints [34.817, 62.968, 17.567, -144.814, 82.241, -185.437]
  Call Extruder(2381.856)
  MoveL 189 to (-26.42, -3.05, 15) mm, rotated rx 180 ry 0 rz -180 deg; joints [34.385, 62.851, 17.923, -145.266, 82.397, -185.241]
  Set speed (130.0 mm/s)
  MoveL 190 to (-41.86, -6.29, 15) mm, rotated rx 180 ry 0 rz -180 deg; joints [35.393, 61.735, 21.432, -144.414, 84.434, -183.97]
  Call Extruder(2386.854)
  Set speed (60.0 mm/s)
  MoveL 191 to (-41.5, -9.47, 15) mm, rotated rx 180 ry 0 rz 180 deg; joints [34.924, 61.623, 21.796, -144.898, 84.609, -183.778]
  Call Extruder(2401.750)
  MoveL 192 to (-38.36, -18.47, 15) mm, rotated rx 180 ry 0 rz -180 deg; joints [33.373, 61.448, 22.374, -146.473, 84.844, -183.408]
  Call Extruder(2416.646)
  MoveL 193 to (-33.28, -26.54, 15) mm, rotated rx -180 ry 0 rz -180 deg; joints [31.763, 61.443, 22.39, -148.088, 84.76, -183.255]
  Call Extruder(2431.541)
  MoveL 194 to (-26.54, -33.29, 15) mm, rotated rx 180 ry 0 rz 180 deg; joints [30.206, 61.608, 21.846, -149.631, 84.346, -183.304]
  Call Extruder(2446.437)
  MoveL 195 to (-18.47, -38.36, 15) mm, rotated rx 180 ry 0 rz -180 deg; joints [28.808, 61.94, 20.769, -150.996, 83.615, -183.528]
  Call Extruder(2461.333)
  MoveL 196 to (-9.47, -41.51, 15) mm, rotated rx 180 ry 0 rz 180 deg; joints [27.654, 62.43, 19.218, -152.094, 82.608, -183.898]
  Call Extruder(2476.229)
  MoveL 197 to (0, -42.57, 15) mm, rotated rx 180 ry 0 rz -180 deg; joints [26.805, 63.065, 17.274, -152.865, 81.386, -184.39]
  Call Extruder(2491.125)
  MoveL 198 to (9.47, -41.5, 15) mm, rotated rx 180 ry 0 rz -180 deg; joints [26.29, 63.822, 15.035, -153.275, 80.022, -184.986]
  Call Extruder(2506.020)
  MoveL 199 to (18.47, -38.36, 15) mm, rotated rx 180 ry 0 rz 180 deg; joints [26.114, 64.671, 12.611, -153.319, 78.598, -185.673]
  Call Extruder(2520.916)
  MoveL 200 to (26.54, -33.28, 15) mm, rotated rx 180 ry 0 rz 180 deg; joints [26.262, 65.571, 10.12, -153.015, 77.195, -186.439]
  Call Extruder(2535.812)
  MoveL 201 to (33.28, -26.54, 15) mm, rotated rx -180 ry 0 rz -180 deg; joints [26.703, 66.477, 7.683, -152.396, 75.887, -187.266]
  Call Extruder(2550.708)
  MoveL 202 to (38.36, -18.47, 15) mm, rotated rx 180 ry 0 rz 180 deg; joints [27.4, 67.341, 5.418, -151.51, 74.744, -188.128]
  Call Extruder(2565.604)
  MoveL 203 to (41.51, -9.47, 15) mm, rotated rx -180 ry 0 rz -180 deg; joints [28.309, 68.111, 3.439, -150.411, 73.822, -188.99]
  Call Extruder(2580.499)
  MoveL 204 to (42.57, 0, 15) mm, rotated rx 180 ry 0 rz -180 deg; joints [29.382, 68.74, 1.848, -149.163, 73.166, -189.809]
  Call Extruder(2595.395)
  MoveL 205 to (41.5, 9.47, 15) mm, rotated rx 180 ry 0 rz 180 deg; joints [30.575, 69.187, 0.73, -147.828, 72.804, -190.535]
  Call Extruder(2610.291)
  MoveL 206 to (38.36, 18.47, 15) mm, rotated rx -180 ry 0 rz 180 deg; joints [31.839, 69.423, 0.145, -146.469, 72.748, -191.118]
  Call Extruder(2625.187)
  MoveL 207 to (33.28, 26.54, 15) mm, rotated rx 180 ry 0 rz 180 deg; joints [33.128, 69.43, 0.128, -145.145, 72.993, -191.514]
  Call Extruder(2640.083)
  MoveL 208 to (26.54, 33.29, 15) mm, rotated rx 180 ry 0 rz 180 deg; joints [34.394, 69.207, 0.68, -143.907, 73.516, -191.688]
  Call Extruder(2654.979)
  MoveL 209 to (18.47, 38.36, 15) mm, rotated rx 180 ry 0 rz -180 deg; joints [35.592, 68.772, 1.768, -142.798, 74.282, -191.62]
  Call Extruder(2669.874)
  MoveL 210 to (9.47, 41.51, 15) mm, rotated rx 180 ry 0 rz -180 deg; joints [36.675, 68.152, 3.334, -141.856, 75.246, -191.31]
  Call Extruder(2684.770)
  MoveL 211 to (0, 42.57, 15) mm, rotated rx 180 ry 0 rz 180 deg; joints [37.594, 67.389, 5.293, -141.114, 76.358, -190.77]
  Call Extruder(2699.666)
  MoveL 212 to (-9.47, 41.51, 15) mm, rotated rx 180 ry 0 rz -180 deg; joints [38.304, 66.53, 7.544, -140.6, 77.565, -190.03]
  Call Extruder(2714.562)
  MoveL 213 to (-18.47, 38.36, 15) mm, rotated rx 180 ry 0 rz 180 deg; joints [38.762, 65.624, 9.974, -140.342, 78.818, -189.133]
  Call Extruder(2729.457)
  MoveL 214 to (-26.54, 33.29, 15) mm, rotated rx 180 ry 0 rz -180 deg; joints [38.928, 64.722, 12.465, -140.364, 80.066, -188.132]
  Call Extruder(2744.353)
  MoveL 215 to (-33.29, 26.54, 15) mm, rotated rx 180 ry 0 rz 180 deg; joints [38.772, 63.87, 14.896, -140.686, 81.264, -187.09]
  Call Extruder(2759.249)
  MoveL 216 to (-38.36, 18.47, 15) mm, rotated rx 180 ry 0 rz 180 deg; joints [38.277, 63.107, 17.149, -141.317, 82.365, -186.072]
  Call Extruder(2774.145)
  MoveL 217 to (-41.51, 9.47, 15) mm, rotated rx 180 ry 0 rz 180 deg; joints [37.447, 62.464, 19.114, -142.253, 83.322, -185.144]
  Call Extruder(2789.041)
  MoveL 218 to (-42.57, 0, 15) mm, rotated rx -180 ry 0 rz 180 deg; joints [36.31, 61.964, 20.69, -143.464, 84.087, -184.365]
  Call Extruder(2796.595)
  MoveL 219 to (-42.03, -4.8, 15) mm, rotated rx -180 ry 0 rz -180 deg; joints [35.612, 61.788, 21.259, -144.188, 84.352, -184.062]
  Set speed (130.0 mm/s)
  MoveL 220 to (-54.1, -7.67, 15) mm, rotated rx 180 ry 0 rz -180 deg; joints [36.421, 60.983, 23.948, -143.472, 85.923, -183.015]
  Call Extruder(2800.668)
  Set speed (30.0 mm/s)
  MoveL 221 to (-53.59, -12.23, 15) mm, rotated rx 180 ry 0 rz 180 deg; joints [35.732, 60.832, 24.472, -144.177, 86.19, -182.746]
  Call Extruder(2811.598)
  MoveL 222 to (-49.52, -23.85, 15) mm, rotated rx 180 ry 0 rz -180 deg; joints [33.663, 60.619, 25.224, -146.268, 86.541, -182.307]
  Call Extruder(2822.528)
  MoveL 223 to (-42.98, -34.27, 15) mm, rotated rx -180 ry 0 rz -180 deg; joints [31.506, 60.613, 25.246, -148.428, 86.47, -182.167]
  Call Extruder(2833.458)
  MoveL 224 to (-34.27, -42.98, 15) mm, rotated rx 180 ry 0 rz 180 deg; joints [29.427, 60.814, 24.536, -150.492, 85.951, -182.288]
  Call Extruder(2844.388)
  MoveL 225 to (-23.85, -49.52, 15) mm, rotated rx 180 ry 0 rz 180 deg; joints [27.581, 61.221, 23.136, -152.305, 85, -182.619]
  Call Extruder(2855.318)
  MoveL 226 to (-12.23, -53.59, 15) mm, rotated rx 180 ry 0 rz 180 deg; joints [26.087, 61.83, 21.123, -153.741, 83.674, -183.111]
  Call Extruder(2866.249)
  MoveL 227 to (0, -54.97, 15) mm, rotated rx -180 ry 0 rz -180 deg; joints [25.019, 62.628, 18.605, -154.722, 82.062, -183.731]
  Call Extruder(2866.680)
  MoveL 228 to (0.48, -54.91, 15) mm, rotated rx -180 ry 0 rz -180 deg; joints [24.994, 62.665, 18.493, -154.743, 81.991, -183.761]
  Call Extruder(2877.179)
  MoveL 229 to (12.23, -53.59, 15) mm, rotated rx 180 ry 0 rz 180 deg; joints [24.406, 63.591, 15.711, -155.214, 80.267, -184.464]
  Call Extruder(2888.109)
  MoveL 230 to (23.85, -49.53, 15) mm, rotated rx 180 ry 0 rz 180 deg; joints [24.239, 64.681, 12.581, -155.222, 78.401, -185.302]
  Call Extruder(2899.039)
  MoveL 231 to (34.27, -42.98, 15) mm, rotated rx 180 ry 0 rz 180 deg; joints [24.487, 65.849, 9.364, -154.777, 76.57, -186.244]
  Call Extruder(2909.969)
  MoveL 232 to (42.98, -34.27, 15) mm, rotated rx -180 ry 0 rz -180 deg; joints [25.101, 67.036, 6.212, -153.931, 74.87, -187.277]
  Call Extruder(2920.900)
  MoveL 233 to (49.52, -23.85, 15) mm, rotated rx 180 ry 0 rz -180 deg; joints [26.025, 68.175, 3.276, -152.75, 73.39, -188.375]
  Call Extruder(2931.830)
  MoveL 234 to (53.59, -12.23, 15) mm, rotated rx 180 ry 0 rz 180 deg; joints [27.2, 69.199, 0.701, -151.309, 72.203, -189.496]
  Call Extruder(2942.760)
  MoveL 235 to (54.97, 0, 15) mm, rotated rx 180 ry 0 rz -180 deg; joints [28.57, 70.04, -1.376, -149.689, 71.365, -190.581]
  Call Extruder(2953.690)
  MoveL 236 to (53.59, 12.23, 15) mm, rotated rx -180 ry 0 rz -180 deg; joints [30.077, 70.641, -2.841, -147.974, 70.916, -191.558]
  Call Extruder(2964.620)
  MoveL 237 to (49.52, 23.85, 15) mm, rotated rx 180 ry 0 rz -180 deg; joints [31.665, 70.959, -3.608, -146.245, 70.867, -192.355]
  Call Extruder(2975.551)
  MoveL 238 to (42.98, 34.27, 15) mm, rotated rx 180 ry 0 rz -180 deg; joints [33.282, 70.968, -3.63, -144.574, 71.21, -192.905]
  Call Extruder(2986.481)
  MoveL 239 to (34.27, 42.98, 15) mm, rotated rx 180 ry 0 rz -180 deg; joints [34.874, 70.668, -2.906, -143.023, 71.912, -193.158]
  Call Extruder(2997.411)
  MoveL 240 to (23.85, 49.53, 15) mm, rotated rx 180 ry 0 rz -180 deg; joints [36.387, 70.083, -1.48, -141.64, 72.92, -193.086]
  Call Extruder(3008.341)
  MoveL 241 to (12.23, 53.59, 15) mm, rotated rx 180 ry 0 rz 180 deg; joints [37.766, 69.254, 0.564, -140.464, 74.173, -192.687]
  Call Extruder(3019.271)
  MoveL 242 to (0, 54.97, 15) mm, rotated rx 180 ry 0 rz 180 deg; joints [38.954, 68.239, 3.113, -139.527, 75.602, -191.979]
  Call Extruder(3030.202)
  MoveL 243 to (-12.23, 53.59, 15) mm, rotated rx -180 ry 0 rz -180 deg; joints [39.895, 67.105, 6.032, -138.862, 77.14, -191.002]
  Call Extruder(3041.132)
  MoveL 244 to (-23.85, 49.53, 15) mm, rotated rx 180 ry 0 rz -180 deg; joints [40.528, 65.919, 9.175, -138.501, 78.725, -189.813]
  Call Extruder(3052.062)
  MoveL 245 to (-34.27, 42.98, 15) mm, rotated rx 180 ry 0 rz 180 deg; joints [40.799, 64.748, 12.392, -138.48, 80.301, -188.484]
  Call Extruder(3062.992)
  MoveL 246 to (-42.98, 34.27, 15) mm, rotated rx -180 ry 0 rz -180 deg; joints [40.659, 63.652, 15.532, -138.833, 81.816, -187.096]
  Call Extruder(3073.923)
  MoveL 247 to (-49.53, 23.85, 15) mm, rotated rx -180 ry 0 rz 180 deg; joints [40.072, 62.68, 18.444, -139.587, 83.22, -185.74]
  Call Extruder(3084.853)
  MoveL 248 to (-53.59, 12.23, 15) mm, rotated rx 180 ry 0 rz 180 deg; joints [39.031, 61.872, 20.988, -140.751, 84.459, -184.511]
  Call Extruder(3095.783)
  MoveL 249 to (-54.97, 0, 15) mm, rotated rx 180 ry 0 rz -180 deg; joints [37.56, 61.251, 23.034, -142.302, 85.472, -183.491]
  Call Extruder(3101.309)
  MoveL 250 to (-54.27, -6.18, 15) mm, rotated rx -180 ry 0 rz -180 deg; joints [36.644, 61.034, 23.773, -143.243, 85.836, -183.105]
  Set speed (130.0 mm/s)
  MoveL 251 to (-49.9, -9.51, 15) mm, rotated rx 180 ry 0 rz 180 deg; joints [35.741, 61.14, 23.409, -144.135, 85.579, -183.19]
  MoveL 252 to (-13.82, -4.91, 15) mm, rotated rx 180 ry 0 rz 180 deg; joints [33.033, 63.638, 15.573, -146.498, 80.971, -185.931]
  Call Extruder(3134.484)
  Set speed (20.0 mm/s)
  MoveL 253 to (-4.92, -13.82, 15) mm, rotated rx 180 ry 0 rz -180 deg; joints [31.126, 63.882, 14.862, -148.379, 80.381, -185.874]
  Call Extruder(3204.290)
  MoveL 254 to (13.82, 4.91, 15) mm, rotated rx -180 ry 0 rz -180 deg; joints [32.046, 66.32, 8.102, -146.982, 76.842, -188.415]
  Call Extruder(3237.465)
  MoveL 255 to (4.91, 13.82, 15) mm, rotated rx 180 ry 0 rz 180 deg; joints [33.834, 66.054, 8.814, -145.225, 77.476, -188.563]
  Set speed (130.0 mm/s)
  MoveL 256 to (4.92, 13.82, 20) mm, rotated rx 180 ry 0 rz 180 deg; joints [33.834, 65.118, 9.367, -145.176, 77.162, -188.787]
  MoveL 257 to (-26.25, -4.54, 20) mm, rotated rx 180 ry 0 rz -180 deg; joints [34.172, 61.809, 18.649, -145.456, 82.117, -185.394]
  Call Extruder(3239.698)
  Set speed (60.0 mm/s)
  MoveL 258 to (-26.09, -5.96, 20) mm, rotated rx 180 ry 0 rz -180 deg; joints [33.969, 61.755, 18.812, -145.668, 82.188, -185.304]
  Call Extruder(3249.063)
  MoveL 259 to (-24.12, -11.61, 20) mm, rotated rx -180 ry 0 rz -180 deg; joints [33.033, 61.635, 19.172, -146.627, 82.303, -185.042]
  Call Extruder(3258.428)
  MoveL 260 to (-20.93, -16.69, 20) mm, rotated rx 180 ry 0 rz 180 deg; joints [32.066, 61.632, 19.182, -147.601, 82.225, -184.907]
  Call Extruder(3267.793)
  MoveL 261 to (-16.69, -20.93, 20) mm, rotated rx -180 ry 0 rz -180 deg; joints [31.126, 61.745, 18.842, -148.529, 81.952, -184.898]
  Call Extruder(3277.158)
  MoveL 262 to (-11.61, -24.11, 20) mm, rotated rx -180 ry 0 rz -180 deg; joints [30.272, 61.97, 18.17, -149.356, 81.494, -185.008]
  Call Extruder(3286.522)
  MoveL 263 to (-5.96, -26.09, 20) mm, rotated rx 180 ry 0 rz 180 deg; joints [29.552, 62.298, 17.199, -150.031, 80.876, -185.224]
  Call Extruder(3295.888)
  MoveL 264 to (0, -26.77, 20) mm, rotated rx 180 ry 0 rz -180 deg; joints [29.003, 62.719, 15.979, -150.519, 80.13, -185.535]
  Call Extruder(3305.253)
  MoveL 265 to (5.96, -26.09, 20) mm, rotated rx 180 ry 0 rz -180 deg; joints [28.65, 63.212, 14.572, -150.794, 79.299, -185.926]
  Call Extruder(3314.617)
  MoveL 266 to (11.61, -24.11, 20) mm, rotated rx 180 ry 0 rz 180 deg; joints [28.503, 63.758, 13.049, -150.85, 78.429, -186.383]
  Call Extruder(3323.982)
  MoveL 267 to (16.69, -20.93, 20) mm, rotated rx -180 ry 0 rz -180 deg; joints [28.559, 64.329, 11.483, -150.689, 77.568, -186.891]
  Call Extruder(3333.348)
  MoveL 268 to (20.93, -16.69, 20) mm, rotated rx -180 ry 0 rz -180 deg; joints [28.808, 64.897, 9.954, -150.328, 76.762, -187.433]
  Call Extruder(3342.712)
  MoveL 269 to (24.11, -11.61, 20) mm, rotated rx -180 ry 0 rz -180 deg; joints [29.229, 65.432, 8.536, -149.793, 76.054, -187.987]
  Call Extruder(3352.077)
  MoveL 270 to (26.09, -5.96, 20) mm, rotated rx 180 ry 0 rz 180 deg; joints [29.796, 65.905, 7.301, -149.115, 75.479, -188.529]
  Call Extruder(3361.442)
  MoveL 271 to (26.77, 0, 20) mm, rotated rx -180 ry 0 rz -180 deg; joints [30.482, 66.288, 6.311, -148.332, 75.065, -189.033]
  Call Extruder(3370.807)
  MoveL 272 to (26.09, 5.96, 20) mm, rotated rx -180 ry 0 rz -180 deg; joints [31.252, 66.558, 5.617, -147.484, 74.83, -189.471]
  Call Extruder(3380.172)
  MoveL 273 to (24.11, 11.61, 20) mm, rotated rx 180 ry 0 rz 180 deg; joints [32.076, 66.7, 5.256, -146.61, 74.783, -189.815]
  Call Extruder(3389.537)
  MoveL 274 to (20.93, 16.69, 20) mm, rotated rx -180 ry 0 rz -180 deg; joints [32.917, 66.704, 5.245, -145.75, 74.923, -190.043]
  Call Extruder(3398.902)
  MoveL 275 to (16.69, 20.93, 20) mm, rotated rx -180 ry 0 rz 180 deg; joints [33.742, 66.57, 5.587, -144.941, 75.239, -190.137]
  Call Extruder(3408.267)
  MoveL 276 to (11.61, 24.12, 20) mm, rotated rx 180 ry 0 rz 180 deg; joints [34.517, 66.307, 6.262, -144.215, 75.71, -190.088]
  Call Extruder(3417.632)
  MoveL 277 to (5.96, 26.09, 20) mm, rotated rx 180 ry 0 rz -180 deg; joints [35.208, 65.93, 7.235, -143.601, 76.312, -189.896]
  Call Extruder(3426.997)
  MoveL 278 to (0, 26.77, 20) mm, rotated rx 180 ry 0 rz -180 deg; joints [35.784, 65.462, 8.457, -143.125, 77.015, -189.568]
  Call Extruder(3436.362)
  MoveL 279 to (-5.96, 26.09, 20) mm, rotated rx 180 ry 0 rz -180 deg; joints [36.214, 64.93, 9.867, -142.808, 77.785, -189.121]
  Call Extruder(3445.727)
  MoveL 280 to (-11.61, 24.12, 20) mm, rotated rx 180 ry 0 rz 180 deg; joints [36.473, 64.363, 11.391, -142.667, 78.587, -188.583]
  Call Extruder(3455.092)
  MoveL 281 to (-16.69, 20.93, 20) mm, rotated rx 180 ry 0 rz 180 deg; joints [36.542, 63.791, 12.957, -142.716, 79.387, -187.982]
  Call Extruder(3464.457)
  MoveL 282 to (-20.93, 16.69, 20) mm, rotated rx 180 ry 0 rz -180 deg; joints [36.407, 63.243, 14.485, -142.959, 80.15, -187.356]
  Call Extruder(3473.822)
  MoveL 283 to (-24.12, 11.61, 20) mm, rotated rx 180 ry 0 rz -180 deg; joints [36.065, 62.746, 15.901, -143.394, 80.844, -186.741]
  Call Extruder(3483.187)
  MoveL 284 to (-26.09, 5.96, 20) mm, rotated rx 180 ry 0 rz 180 deg; joints [35.528, 62.321, 17.133, -144.009, 81.434, -186.174]
  Call Extruder(3492.552)
  MoveL 285 to (-26.77, 0, 20) mm, rotated rx 180 ry 0 rz 180 deg; joints [34.817, 61.986, 18.12, -144.78, 81.891, -185.687]
  Call Extruder(3497.341)
  MoveL 286 to (-26.42, -3.05, 20) mm, rotated rx -180 ry 0 rz -180 deg; joints [34.385, 61.867, 18.477, -145.233, 82.043, -185.489]
  Set speed (130.0 mm/s)
  MoveL 287 to (-41.86, -6.29, 20) mm, rotated rx 180 ry 0 rz 180 deg; joints [35.393, 60.727, 21.99, -144.387, 84.068, -184.233]
  Call Extruder(3502.339)
  Set speed (60.0 mm/s)
  MoveL 288 to (-41.5, -9.47, 20) mm, rotated rx 180 ry 0 rz 180 deg; joints [34.924, 60.613, 22.355, -144.873, 84.239, -184.04]
  Call Extruder(3517.234)
  MoveL 289 to (-38.36, -18.47, 20) mm, rotated rx 180 ry 0 rz -180 deg; joints [33.373, 60.434, 22.933, -146.45, 84.464, -183.66]
  Call Extruder(3532.130)
  MoveL 290 to (-33.29, -26.54, 20) mm, rotated rx -180 ry 0 rz 180 deg; joints [31.763, 60.429, 22.95, -148.065, 84.374, -183.497]
  Call Extruder(3547.026)
  MoveL 291 to (-26.54, -33.28, 20) mm, rotated rx -180 ry 0 rz -180 deg; joints [30.206, 60.597, 22.404, -149.607, 83.956, -183.534]
  Call Extruder(3561.922)
  MoveL 292 to (-18.47, -38.36, 20) mm, rotated rx 180 ry 0 rz -180 deg; joints [28.808, 60.937, 21.326, -150.971, 83.225, -183.746]
  Call Extruder(3576.817)
  MoveL 293 to (-9.47, -41.5, 20) mm, rotated rx 180 ry 0 rz -180 deg; joints [27.654, 61.438, 19.773, -152.067, 82.221, -184.105]
  Call Extruder(3591.713)
  MoveL 294 to (0, -42.57, 20) mm, rotated rx 180 ry 0 rz 180 deg; joints [26.805, 62.085, 17.827, -152.834, 81.006, -184.587]
  Call Extruder(3606.609)
  MoveL 295 to (9.47, -41.5, 20) mm, rotated rx -180 ry 0 rz -180 deg; joints [26.29, 62.855, 15.587, -153.241, 79.652, -185.176]
  Call Extruder(3621.505)
  MoveL 296 to (18.47, -38.36, 20) mm, rotated rx -180 ry 0 rz 180 deg; joints [26.114, 63.717, 13.163, -153.282, 78.239, -185.858]
  Call Extruder(3636.401)
  MoveL 297 to (26.54, -33.28, 20) mm, rotated rx 180 ry 0 rz -180 deg; joints [26.262, 64.629, 10.672, -152.974, 76.847, -186.621]
  Call Extruder(3651.297)
  MoveL 298 to (33.28, -26.54, 20) mm, rotated rx -180 ry 0 rz 180 deg; joints [26.703, 65.546, 8.237, -152.352, 75.553, -187.446]
  Call Extruder(3666.192)
  MoveL 299 to (38.36, -18.47, 20) mm, rotated rx 180 ry 0 rz 180 deg; joints [27.4, 66.419, 5.974, -151.461, 74.422, -188.309]
  Call Extruder(3681.088)
  MoveL 300 to (41.5, -9.47, 20) mm, rotated rx 180 ry 0 rz 180 deg; joints [28.309, 67.196, 3.998, -150.359, 73.512, -189.174]
  Call Extruder(3695.984)
  MoveL 301 to (42.57, 0, 20) mm, rotated rx 180 ry 0 rz -180 deg; joints [29.382, 67.83, 2.41, -149.108, 72.867, -189.996]
  Call Extruder(3710.880)
  MoveL 302 to (41.5, 9.47, 20) mm, rotated rx 180 ry 0 rz -180 deg; joints [30.575, 68.281, 1.294, -147.771, 72.514, -190.726]
  Call Extruder(3725.775)
  MoveL 303 to (38.36, 18.47, 20) mm, rotated rx 180 ry 0 rz -180 deg; joints [31.839, 68.518, 0.711, -146.41, 72.465, -191.315]
  Call Extruder(3740.671)
  MoveL 304 to (33.28, 26.54, 20) mm, rotated rx 180 ry 0 rz -180 deg; joints [33.128, 68.524, 0.694, -145.085, 72.714, -191.717]
  Call Extruder(3755.567)
  MoveL 305 to (26.54, 33.29, 20) mm, rotated rx -180 ry 0 rz -180 deg; joints [34.394, 68.301, 1.244, -143.847, 73.239, -191.898]
  Call Extruder(3770.463)
  MoveL 306 to (18.47, 38.36, 20) mm, rotated rx 180 ry 0 rz 180 deg; joints [35.592, 67.862, 2.33, -142.738, 74.005, -191.839]
  Call Extruder(3785.359)
  MoveL 307 to (9.47, 41.51, 20) mm, rotated rx 180 ry 0 rz 180 deg; joints [36.675, 67.238, 3.893, -141.798, 74.966, -191.537]
  Call Extruder(3800.255)
  MoveL 308 to (0, 42.57, 20) mm, rotated rx -180 ry 0 rz -180 deg; joints [37.594, 66.468, 5.849, -141.058, 76.073, -191.006]
  Call Extruder(3815.150)
  MoveL 309 to (-9.47, 41.51, 20) mm, rotated rx 180 ry 0 rz 180 deg; joints [38.304, 65.599, 8.098, -140.547, 77.274, -190.275]
  Call Extruder(3830.046)
  MoveL 310 to (-18.47, 38.36, 20) mm, rotated rx 180 ry 0 rz -180 deg; joints [38.762, 64.683, 10.527, -140.292, 78.518, -189.386]
  Call Extruder(3844.942)
  MoveL 311 to (-26.54, 33.29, 20) mm, rotated rx 180 ry 0 rz -180 deg; joints [38.928, 63.769, 13.017, -140.318, 79.757, -188.393]
  Call Extruder(3859.838)
  MoveL 312 to (-33.29, 26.54, 20) mm, rotated rx 180 ry 0 rz 180 deg; joints [38.772, 62.904, 15.448, -140.645, 80.943, -187.356]
  Call Extruder(3874.734)
  MoveL 313 to (-38.36, 18.47, 20) mm, rotated rx 180 ry 0 rz 180 deg; joints [38.277, 62.127, 17.703, -141.281, 82.032, -186.341]
  Call Extruder(3889.629)
  MoveL 314 to (-41.51, 9.47, 20) mm, rotated rx 180 ry 0 rz 180 deg; joints [37.447, 61.472, 19.669, -142.221, 82.977, -185.414]
  Call Extruder(3904.525)
  MoveL 315 to (-42.57, 0, 20) mm, rotated rx 180 ry 0 rz -180 deg; joints [36.31, 60.962, 21.247, -143.436, 83.729, -184.632]
  Call Extruder(3912.079)
  MoveL 316 to (-42.03, -4.8, 20) mm, rotated rx 180 ry 0 rz -180 deg; joints [35.612, 60.781, 21.816, -144.161, 83.988, -184.326]
  Set speed (130.0 mm/s)
  MoveL 317 to (-54.1, -7.67, 20) mm, rotated rx 180 ry 0 rz -180 deg; joints [36.421, 59.957, 24.51, -143.451, 85.55, -183.292]
  Call Extruder(3916.152)
  Set speed (30.0 mm/s)
  MoveL 318 to (-53.59, -12.23, 20) mm, rotated rx -180 ry 0 rz 180 deg; joints [35.732, 59.801, 25.036, -144.158, 85.811, -183.02]
  Call Extruder(3927.082)
  MoveL 319 to (-49.53, -23.85, 20) mm, rotated rx 180 ry 0 rz -180 deg; joints [33.663, 59.582, 25.789, -146.251, 86.149, -182.569]
  Call Extruder(3938.012)
  MoveL 320 to (-42.98, -34.27, 20) mm, rotated rx 180 ry 0 rz -180 deg; joints [31.506, 59.576, 25.811, -148.412, 86.068, -182.414]
  Call Extruder(3948.943)
  MoveL 321 to (-34.27, -42.98, 20) mm, rotated rx -180 ry 0 rz -180 deg; joints [29.427, 59.783, 25.1, -150.475, 85.544, -182.519]
  Call Extruder(3959.873)
  MoveL 322 to (-23.85, -49.52, 20) mm, rotated rx 180 ry 0 rz 180 deg; joints [27.581, 60.201, 23.697, -152.286, 84.593, -182.834]
  Call Extruder(3970.803)
  MoveL 323 to (-12.23, -53.59, 20) mm, rotated rx 180 ry 0 rz 180 deg; joints [26.087, 60.824, 21.681, -153.719, 83.272, -183.311]
  Call Extruder(3981.733)
  MoveL 324 to (0, -54.97, 20) mm, rotated rx 180 ry 0 rz -180 deg; joints [25.019, 61.639, 19.16, -154.696, 81.669, -183.919]
  Call Extruder(3982.538)
  MoveL 325 to (0.9, -54.87, 20) mm, rotated rx -180 ry 0 rz -180 deg; joints [24.972, 61.709, 18.95, -154.734, 81.539, -183.973]
  Call Extruder(3992.663)
  MoveL 326 to (12.23, -53.59, 20) mm, rotated rx -180 ry 0 rz 180 deg; joints [24.406, 62.62, 16.263, -155.184, 79.887, -184.642]
  Call Extruder(4003.594)
  MoveL 327 to (23.85, -49.52, 20) mm, rotated rx -180 ry 0 rz -180 deg; joints [24.239, 63.727, 13.132, -155.187, 78.036, -185.475]
  Call Extruder(4014.524)
  MoveL 328 to (34.27, -42.98, 20) mm, rotated rx -180 ry 0 rz 180 deg; joints [24.487, 64.911, 9.917, -154.737, 76.221, -186.413]
  Call Extruder(4025.454)
  MoveL 329 to (42.98, -34.27, 20) mm, rotated rx -180 ry 0 rz 180 deg; joints [25.101, 66.111, 6.767, -153.887, 74.538, -187.445]
  Call Extruder(4036.384)
  MoveL 330 to (49.52, -23.85, 20) mm, rotated rx 180 ry 0 rz -180 deg; joints [26.025, 67.261, 3.835, -152.701, 73.074, -188.545]
  Call Extruder(4047.314)
  MoveL 331 to (53.59, -12.23, 20) mm, rotated rx 180 ry 0 rz -180 deg; joints [27.2, 68.292, 1.265, -151.256, 71.902, -189.669]
  Call Extruder(4058.245)
  MoveL 332 to (54.97, 0, 20) mm, rotated rx -180 ry 0 rz -180 deg; joints [28.57, 69.139, -0.807, -149.632, 71.079, -190.758]
  Call Extruder(4069.175)
  MoveL 333 to (53.59, 12.23, 20) mm, rotated rx 180 ry 0 rz 180 deg; joints [30.077, 69.744, -2.268, -147.914, 70.64, -191.741]
  Call Extruder(4080.105)
  MoveL 334 to (49.52, 23.85, 20) mm, rotated rx 180 ry 0 rz 180 deg; joints [31.665, 70.062, -3.033, -146.182, 70.6, -192.544]
  Call Extruder(4091.035)
  MoveL 335 to (42.98, 34.27, 20) mm, rotated rx 180 ry 0 rz 180 deg; joints [33.282, 70.072, -3.055, -144.51, 70.949, -193.102]
  Call Extruder(4101.965)
  MoveL 336 to (34.27, 42.98, 20) mm, rotated rx 180 ry 0 rz 180 deg; joints [34.874, 69.771, -2.333, -142.958, 71.652, -193.364]
  Call Extruder(4112.896)
  MoveL 337 to (23.85, 49.53, 20) mm, rotated rx 180 ry 0 rz -180 deg; joints [36.387, 69.182, -0.911, -141.576, 72.66, -193.302]
  Call Extruder(4123.826)
  MoveL 338 to (12.23, 53.59, 20) mm, rotated rx 180 ry 0 rz 180 deg; joints [37.766, 68.348, 1.128, -140.401, 73.91, -192.913]
  Call Extruder(4134.756)
  MoveL 339 to (0, 54.97, 20) mm, rotated rx 180 ry 0 rz 180 deg; joints [38.954, 67.325, 3.672, -139.467, 75.333, -192.216]
  Call Extruder(4145.686)
  MoveL 340 to (-12.23, 53.59, 20) mm, rotated rx 180 ry 0 rz 180 deg; joints [39.895, 66.181, 6.587, -138.806, 76.863, -191.251]
  Call Extruder(4156.616)
  MoveL 341 to (-23.85, 49.53, 20) mm, rotated rx 180 ry 0 rz -180 deg; joints [40.528, 64.982, 9.728, -138.449, 78.437, -190.074]
  Call Extruder(4167.547)
  MoveL 342 to (-34.27, 42.98, 20) mm, rotated rx 180 ry 0 rz 180 deg; joints [40.799, 63.796, 12.944, -138.434, 80.001, -188.754]
  Call Extruder(4178.477)
  MoveL 343 to (-42.98, 34.27, 20) mm, rotated rx -180 ry 0 rz -180 deg; joints [40.659, 62.682, 16.084, -138.793, 81.501, -187.374]
  Call Extruder(4189.407)
  MoveL 344 to (-49.53, 23.85, 20) mm, rotated rx 180 ry 0 rz 180 deg; joints [40.072, 61.693, 18.999, -139.553, 82.89, -186.024]
  Call Extruder(4200.337)
  MoveL 345 to (-53.59, 12.23, 20) mm, rotated rx 180 ry 0 rz -180 deg; joints [39.031, 60.867, 21.545, -140.723, 84.113, -184.795]
  Call Extruder(4211.267)
  MoveL 346 to (-54.97, 0, 20) mm, rotated rx -180 ry 0 rz -180 deg; joints [37.56, 60.232, 23.594, -142.279, 85.109, -183.773]
  Call Extruder(4216.793)
  MoveL 347 to (-54.27, -6.18, 20) mm, rotated rx 180 ry 0 rz -180 deg; joints [36.644, 60.009, 24.335, -143.222, 85.465, -183.383]
  Set speed (130.0 mm/s)
  MoveL 348 to (-49.9, -9.51, 20) mm, rotated rx 180 ry 0 rz -180 deg; joints [35.741, 60.118, 23.971, -144.114, 85.205, -183.461]
  MoveL 349 to (-4.92, 13.82, 20) mm, rotated rx 180 ry 0 rz 180 deg; joints [34.648, 64.31, 11.534, -144.521, 78.394, -188.16]
  Call Extruder(4249.968)
  Set speed (20.0 mm/s)
  MoveL 350 to (-13.82, 4.91, 20) mm, rotated rx 180 ry 0 rz 180 deg; joints [34.301, 63.151, 14.744, -145.097, 80.025, -186.891]
  Call Extruder(4319.775)
  MoveL 351 to (4.91, -13.82, 20) mm, rotated rx 180 ry 0 rz 180 deg; joints [30.357, 63.685, 13.249, -148.984, 78.751, -186.689]
  Call Extruder(4352.950)
  MoveL 352 to (13.82, -4.91, 20) mm, rotated rx 180 ry 0 rz -180 deg; joints [30.824, 64.866, 10.038, -148.284, 77.076, -187.87]
  Set speed (130.0 mm/s)
  MoveL 353 to (13.82, -4.91, 25) mm, rotated rx 180 ry 0 rz 180 deg; joints [30.824, 63.931, 10.573, -148.235, 76.736, -188.086]
  MoveL 354 to (-26.25, -4.54, 25) mm, rotated rx 180 ry 0 rz -180 deg; joints [34.172, 60.826, 19.186, -145.42, 81.75, -185.649]
  Call Extruder(4355.182)
  Set speed (60.0 mm/s)
  MoveL 355 to (-26.09, -5.96, 25) mm, rotated rx 180 ry 0 rz 180 deg; joints [33.969, 60.771, 19.349, -145.633, 81.819, -185.558]
  Call Extruder(4364.547)
  MoveL 356 to (-24.12, -11.61, 25) mm, rotated rx 180 ry 0 rz 180 deg; joints [33.033, 60.649, 19.71, -146.593, 81.928, -185.291]
  Call Extruder(4373.912)
  MoveL 357 to (-20.93, -16.69, 25) mm, rotated rx 180 ry 0 rz -180 deg; joints [32.066, 60.645, 19.72, -147.567, 81.846, -185.15]
  Call Extruder(4383.277)
  MoveL 358 to (-16.69, -20.93, 25) mm, rotated rx 180 ry 0 rz -180 deg; joints [31.126, 60.76, 19.38, -148.495, 81.571, -185.134]
  Call Extruder(4392.642)
  MoveL 359 to (-11.61, -24.11, 25) mm, rotated rx 180 ry 0 rz -180 deg; joints [30.272, 60.989, 18.706, -149.321, 81.113, -185.236]
  Call Extruder(4402.007)
  MoveL 360 to (-5.96, -26.09, 25) mm, rotated rx 180 ry 0 rz 180 deg; joints [29.552, 61.325, 17.735, -149.995, 80.497, -185.446]
  Call Extruder(4411.372)
  MoveL 361 to (0, -26.77, 25) mm, rotated rx 180 ry 0 rz -180 deg; joints [29.003, 61.752, 16.514, -150.481, 79.755, -185.751]
  Call Extruder(4420.737)
  MoveL 362 to (5.96, -26.09, 25) mm, rotated rx 180 ry 0 rz -180 deg; joints [28.65, 62.254, 15.107, -150.755, 78.929, -186.137]
  Call Extruder(4430.102)
  MoveL 363 to (11.61, -24.11, 25) mm, rotated rx 180 ry 0 rz -180 deg; joints [28.503, 62.808, 13.583, -150.808, 78.066, -186.59]
  Call Extruder(4439.467)
  MoveL 364 to (16.69, -20.93, 25) mm, rotated rx 180 ry 0 rz -180 deg; joints [28.559, 63.387, 12.018, -150.645, 77.213, -187.096]
  Call Extruder(4448.832)
  MoveL 365 to (20.93, -16.69, 25) mm, rotated rx -180 ry 0 rz 180 deg; joints [28.808, 63.963, 10.489, -150.281, 76.416, -187.636]
  Call Extruder(4458.197)
  MoveL 366 to (24.11, -11.61, 25) mm, rotated rx 180 ry 0 rz 180 deg; joints [29.229, 64.504, 9.072, -149.743, 75.715, -188.191]
  Call Extruder(4467.562)
  MoveL 367 to (26.09, -5.96, 25) mm, rotated rx 180 ry 0 rz 180 deg; joints [29.796, 64.982, 7.838, -149.063, 75.148, -188.734]
  Call Extruder(4476.927)
  MoveL 368 to (26.77, 0, 25) mm, rotated rx -180 ry 0 rz -180 deg; joints [30.482, 65.369, 6.849, -148.278, 74.741, -189.24]
  Call Extruder(4486.292)
  MoveL 369 to (26.09, 5.96, 25) mm, rotated rx 180 ry 0 rz 180 deg; joints [31.252, 65.642, 6.156, -147.428, 74.512, -189.681]
  Call Extruder(4495.657)
  MoveL 370 to (24.11, 11.61, 25) mm, rotated rx 180 ry 0 rz -180 deg; joints [32.076, 65.785, 5.795, -146.553, 74.47, -190.029]
  Call Extruder(4505.022)
  MoveL 371 to (20.93, 16.69, 25) mm, rotated rx 180 ry 0 rz -180 deg; joints [32.917, 65.789, 5.785, -145.693, 74.613, -190.262]
  Call Extruder(4514.387)
  MoveL 372 to (16.69, 20.93, 25) mm, rotated rx 180 ry 0 rz -180 deg; joints [33.742, 65.654, 6.125, -144.883, 74.93, -190.362]
  Call Extruder(4523.752)
  MoveL 373 to (11.61, 24.12, 25) mm, rotated rx -180 ry 0 rz 180 deg; joints [34.517, 65.389, 6.8, -144.157, 75.402, -190.318]
  Call Extruder(4533.117)
  MoveL 374 to (5.96, 26.09, 25) mm, rotated rx 180 ry 0 rz 180 deg; joints [35.208, 65.008, 7.772, -143.545, 76.002, -190.131]
  Call Extruder(4542.482)
  MoveL 375 to (0, 26.77, 25) mm, rotated rx 180 ry 0 rz 180 deg; joints [35.784, 64.535, 8.993, -143.07, 76.702, -189.809]
  Call Extruder(4551.847)
  MoveL 376 to (-5.96, 26.09, 25) mm, rotated rx 180 ry 0 rz 180 deg; joints [36.214, 63.996, 10.402, -142.755, 77.467, -189.368]
  Call Extruder(4561.212)
  MoveL 377 to (-11.61, 24.12, 25) mm, rotated rx -180 ry 0 rz 180 deg; joints [36.473, 63.421, 11.926, -142.617, 78.264, -188.834]
  Call Extruder(4570.576)
  MoveL 378 to (-16.69, 20.93, 25) mm, rotated rx 180 ry 0 rz 180 deg; joints [36.542, 62.841, 13.491, -142.668, 79.057, -188.238]
  Call Extruder(4579.942)
  MoveL 379 to (-20.93, 16.69, 25) mm, rotated rx 180 ry 0 rz -180 deg; joints [36.407, 62.285, 15.02, -142.914, 79.813, -187.615]
  Call Extruder(4589.307)
  MoveL 380 to (-24.12, 11.61, 25) mm, rotated rx -180 ry 0 rz -180 deg; joints [36.065, 61.78, 16.436, -143.352, 80.498, -187.002]
  Call Extruder(4598.671)
  MoveL 381 to (-26.09, 5.96, 25) mm, rotated rx 180 ry 0 rz -180 deg; joints [35.528, 61.347, 17.669, -143.97, 81.08, -186.435]
  Call Extruder(4608.037)
  MoveL 382 to (-26.77, 0, 25) mm, rotated rx 180 ry 0 rz -180 deg; joints [34.817, 61.006, 18.657, -144.742, 81.529, -185.945]
  Call Extruder(4612.825)
  MoveL 383 to (-26.42, -3.05, 25) mm, rotated rx -180 ry 0 rz -180 deg; joints [34.385, 60.884, 19.014, -145.197, 81.677, -185.745]
  Set speed (130.0 mm/s)
  MoveL 384 to (-41.86, -6.3, 25) mm, rotated rx 180 ry 0 rz 180 deg; joints [35.393, 59.72, 22.532, -144.358, 83.69, -184.506]
  Call Extruder(4617.823)
  Set speed (60.0 mm/s)
  MoveL 385 to (-41.51, -9.47, 25) mm, rotated rx 180 ry 0 rz -180 deg; joints [34.924, 59.604, 22.897, -144.845, 83.857, -184.31]
  Call Extruder(4632.719)
  MoveL 386 to (-38.36, -18.47, 25) mm, rotated rx -180 ry 0 rz 180 deg; joints [33.373, 59.42, 23.476, -146.424, 84.072, -183.922]
  Call Extruder(4647.615)
  MoveL 387 to (-33.29, -26.54, 25) mm, rotated rx -180 ry 0 rz -180 deg; joints [31.763, 59.415, 23.493, -148.04, 83.974, -183.747]
  Call Extruder(4662.510)
  MoveL 388 to (-26.54, -33.28, 25) mm, rotated rx -180 ry 0 rz -180 deg; joints [30.206, 59.588, 22.946, -149.582, 83.553, -183.772]
  Call Extruder(4677.406)
  MoveL 389 to (-18.47, -38.36, 25) mm, rotated rx 180 ry 0 rz 180 deg; joints [28.808, 59.935, 21.867, -150.943, 82.822, -183.971]
  Call Extruder(4692.302)
  MoveL 390 to (-9.47, -41.51, 25) mm, rotated rx 180 ry 0 rz 180 deg; joints [27.654, 60.447, 20.312, -152.037, 81.822, -184.319]
  Call Extruder(4707.198)
  MoveL 391 to (0, -42.57, 25) mm, rotated rx 180 ry 0 rz 180 deg; joints [26.805, 61.107, 18.364, -152.802, 80.613, -184.791]
  Call Extruder(4722.094)
  MoveL 392 to (9.47, -41.5, 25) mm, rotated rx 180 ry 0 rz -180 deg; joints [26.29, 61.891, 16.122, -153.205, 79.269, -185.372]
  Call Extruder(4736.989)
  MoveL 393 to (18.47, -38.36, 25) mm, rotated rx 180 ry 0 rz 180 deg; joints [26.114, 62.766, 13.697, -153.243, 77.867, -186.049]
  Call Extruder(4751.885)
  MoveL 394 to (26.54, -33.28, 25) mm, rotated rx 180 ry 0 rz 180 deg; joints [26.262, 63.691, 11.207, -152.931, 76.489, -186.809]
  Call Extruder(4766.781)
  MoveL 395 to (33.28, -26.54, 25) mm, rotated rx 180 ry 0 rz -180 deg; joints [26.703, 64.62, 8.773, -152.304, 75.207, -187.634]
  Call Extruder(4781.677)
  MoveL 396 to (38.36, -18.47, 25) mm, rotated rx -180 ry 0 rz -180 deg; joints [27.4, 65.501, 6.513, -151.41, 74.089, -188.497]
  Call Extruder(4796.572)
  MoveL 397 to (41.5, -9.47, 25) mm, rotated rx 180 ry 0 rz 180 deg; joints [28.309, 66.286, 4.539, -150.305, 73.192, -189.364]
  Call Extruder(4811.468)
  MoveL 398 to (42.57, 0, 25) mm, rotated rx 180 ry 0 rz 180 deg; joints [29.382, 66.926, 2.953, -149.05, 72.557, -190.19]
  Call Extruder(4826.364)
  MoveL 399 to (41.5, 9.47, 25) mm, rotated rx 180 ry 0 rz -180 deg; joints [30.575, 67.379, 1.839, -147.71, 72.213, -190.926]
  Call Extruder(4841.260)
  MoveL 400 to (38.36, 18.47, 25) mm, rotated rx 180 ry 0 rz 180 deg; joints [31.839, 67.618, 1.257, -146.348, 72.171, -191.52]
  Call Extruder(4856.156)
  MoveL 401 to (33.28, 26.54, 25) mm, rotated rx 180 ry 0 rz 180 deg; joints [33.128, 67.625, 1.24, -145.022, 72.425, -191.929]
  Call Extruder(4871.052)
  MoveL 402 to (26.54, 33.29, 25) mm, rotated rx 180 ry 0 rz -180 deg; joints [34.394, 67.4, 1.789, -143.783, 72.952, -192.118]
  Call Extruder(4885.947)
  MoveL 403 to (18.47, 38.36, 25) mm, rotated rx 180 ry 0 rz 180 deg; joints [35.592, 66.958, 2.874, -142.675, 73.718, -192.067]
  Call Extruder(4900.843)
  MoveL 404 to (9.47, 41.51, 25) mm, rotated rx 180 ry 0 rz -180 deg; joints [36.675, 66.328, 4.434, -141.736, 74.677, -191.774]
  Call Extruder(4915.739)
  MoveL 405 to (0, 42.57, 25) mm, rotated rx -180 ry 0 rz 180 deg; joints [37.594, 65.551, 6.388, -140.998, 75.779, -191.252]
  Call Extruder(4930.635)
  MoveL 406 to (-9.47, 41.51, 25) mm, rotated rx 180 ry 0 rz -180 deg; joints [38.304, 64.673, 8.634, -140.49, 76.973, -190.53]
  Call Extruder(4945.530)
  MoveL 407 to (-18.47, 38.36, 25) mm, rotated rx 180 ry 0 rz 180 deg; joints [38.762, 63.746, 11.061, -140.239, 78.209, -189.649]
  Call Extruder(4960.426)
  MoveL 408 to (-26.54, 33.28, 25) mm, rotated rx -180 ry 0 rz -180 deg; joints [38.928, 62.819, 13.551, -140.269, 79.437, -188.663]
  Call Extruder(4975.322)
  MoveL 409 to (-33.29, 26.54, 25) mm, rotated rx 180 ry 0 rz -180 deg; joints [38.772, 61.94, 15.983, -140.6, 80.612, -187.631]
  Call Extruder(4990.218)
  MoveL 410 to (-38.36, 18.47, 25) mm, rotated rx 180 ry 0 rz 180 deg; joints [38.277, 61.15, 18.239, -141.241, 81.689, -186.62]
  Call Extruder(5005.114)
  MoveL 411 to (-41.51, 9.47, 25) mm, rotated rx -180 ry 0 rz 180 deg; joints [37.447, 60.482, 20.207, -142.186, 82.62, -185.693]
  Call Extruder(5020.010)
  MoveL 412 to (-42.57, 0, 25) mm, rotated rx -180 ry 0 rz 180 deg; joints [36.31, 59.961, 21.788, -143.405, 83.359, -184.908]
  Call Extruder(5027.564)
  MoveL 413 to (-42.03, -4.8, 25) mm, rotated rx 180 ry 0 rz 180 deg; joints [35.612, 59.776, 22.358, -144.131, 83.612, -184.599]
  Set speed (130.0 mm/s)
  MoveL 414 to (-54.1, -7.67, 25) mm, rotated rx -180 ry 0 rz 180 deg; joints [36.421, 58.931, 25.056, -143.428, 85.165, -183.578]
  Call Extruder(5031.636)
  Set speed (30.0 mm/s)
  MoveL 415 to (-53.59, -12.23, 25) mm, rotated rx 180 ry 0 rz 180 deg; joints [35.732, 58.772, 25.583, -144.136, 85.42, -183.304]
  Call Extruder(5042.567)
  MoveL 416 to (-49.53, -23.85, 25) mm, rotated rx -180 ry 0 rz -180 deg; joints [33.663, 58.546, 26.338, -146.232, 85.744, -182.841]
  Call Extruder(5053.497)
  MoveL 417 to (-42.98, -34.27, 25) mm, rotated rx -180 ry 0 rz 180 deg; joints [31.506, 58.54, 26.36, -148.393, 85.653, -182.671]
  Call Extruder(5064.427)
  MoveL 418 to (-34.27, -42.98, 25) mm, rotated rx -180 ry 0 rz 180 deg; joints [29.427, 58.752, 25.647, -150.456, 85.124, -182.758]
  Call Extruder(5075.357)
  MoveL 419 to (-23.85, -49.53, 25) mm, rotated rx 180 ry 0 rz 180 deg; joints [27.581, 59.181, 24.241, -152.264, 84.173, -183.056]
  Call Extruder(5086.287)
  MoveL 420 to (-12.23, -53.59, 25) mm, rotated rx 180 ry 0 rz 180 deg; joints [26.087, 59.82, 22.222, -153.694, 82.857, -183.518]
  Call Extruder(5097.218)
  MoveL 421 to (0, -54.97, 25) mm, rotated rx -180 ry 0 rz 180 deg; joints [25.019, 60.653, 19.698, -154.667, 81.263, -184.113]
  Call Extruder(5098.395)
  MoveL 422 to (1.32, -54.82, 25) mm, rotated rx 180 ry 0 rz 180 deg; joints [24.951, 60.757, 19.39, -154.722, 81.074, -184.191]
  Call Extruder(5108.148)
  MoveL 423 to (12.23, -53.59, 25) mm, rotated rx -180 ry 0 rz -180 deg; joints [24.406, 61.652, 16.799, -155.15, 79.495, -184.826]
  Call Extruder(5119.078)
  MoveL 424 to (23.85, -49.52, 25) mm, rotated rx 180 ry 0 rz 180 deg; joints [24.239, 62.777, 13.667, -155.149, 77.659, -185.653]
  Call Extruder(5130.008)
  MoveL 425 to (34.27, -42.98, 25) mm, rotated rx -180 ry 0 rz -180 deg; joints [24.487, 63.977, 10.452, -154.695, 75.86, -186.589]
  Call Extruder(5140.938)
  MoveL 426 to (42.98, -34.27, 25) mm, rotated rx -180 ry 0 rz 180 deg; joints [25.101, 65.19, 7.305, -153.839, 74.194, -187.621]
  Call Extruder(5151.869)
  MoveL 427 to (49.52, -23.85, 25) mm, rotated rx -180 ry 0 rz -180 deg; joints [26.025, 66.351, 4.376, -152.649, 72.747, -188.722]
  Call Extruder(5162.799)
  MoveL 428 to (53.59, -12.23, 25) mm, rotated rx -180 ry 0 rz -180 deg; joints [27.2, 67.391, 1.811, -151.2, 71.59, -189.85]
  Call Extruder(5173.729)
  MoveL 429 to (54.97, 0, 25) mm, rotated rx 180 ry 0 rz -180 deg; joints [28.57, 68.244, -0.257, -149.572, 70.781, -190.943]
  Call Extruder(5184.659)
  MoveL 430 to (53.59, 12.23, 25) mm, rotated rx 180 ry 0 rz 180 deg; joints [30.077, 68.852, -1.715, -147.85, 70.354, -191.932]
  Call Extruder(5195.589)
  MoveL 431 to (49.52, 23.85, 25) mm, rotated rx 180 ry 0 rz -180 deg; joints [31.665, 69.172, -2.477, -146.116, 70.322, -192.742]
  Call Extruder(5206.520)
  MoveL 432 to (42.98, 34.27, 25) mm, rotated rx 180 ry 0 rz 180 deg; joints [33.282, 69.182, -2.499, -144.442, 70.676, -193.308]
  Call Extruder(5217.450)
  MoveL 433 to (34.27, 42.98, 25) mm, rotated rx 180 ry 0 rz 180 deg; joints [34.874, 68.879, -1.779, -142.89, 71.383, -193.579]
  Call Extruder(5228.380)
  MoveL 434 to (23.85, 49.53, 25) mm, rotated rx 180 ry 0 rz -180 deg; joints [36.387, 68.287, -0.361, -141.508, 72.39, -193.527]
  Call Extruder(5239.310)
  MoveL 435 to (12.23, 53.59, 25) mm, rotated rx 180 ry 0 rz 180 deg; joints [37.766, 67.447, 1.674, -140.335, 73.636, -193.149]
  Call Extruder(5250.240)
  MoveL 436 to (0, 54.97, 25) mm, rotated rx 180 ry 0 rz -180 deg; joints [38.954, 66.417, 4.214, -139.404, 75.053, -192.464]
  Call Extruder(5261.171)
  MoveL 437 to (-12.23, 53.59, 25) mm, rotated rx 180 ry 0 rz -180 deg; joints [39.895, 65.261, 7.125, -138.746, 76.575, -191.51]
  Call Extruder(5272.101)
  MoveL 438 to (-23.85, 49.52, 25) mm, rotated rx 180 ry 0 rz 180 deg; joints [40.528, 64.048, 10.263, -138.394, 78.139, -190.343]
  Call Extruder(5283.031)
  MoveL 439 to (-34.27, 42.98, 25) mm, rotated rx 180 ry 0 rz -180 deg; joints [40.799, 62.846, 13.479, -138.384, 79.69, -189.034]
  Call Extruder(5293.961)
  MoveL 440 to (-42.98, 34.27, 25) mm, rotated rx 180 ry 0 rz 180 deg; joints [40.659, 61.715, 16.619, -138.749, 81.177, -187.662]
  Call Extruder(5304.891)
  MoveL 441 to (-49.53, 23.85, 25) mm, rotated rx 180 ry 0 rz -180 deg; joints [40.072, 60.707, 19.536, -139.516, 82.549, -186.317]
  Call Extruder(5315.822)
  MoveL 442 to (-53.59, 12.23, 25) mm, rotated rx 180 ry 0 rz -180 deg; joints [39.031, 59.864, 22.086, -140.691, 83.755, -185.09]
  Call Extruder(5326.752)
  MoveL 443 to (-54.97, 0, 25) mm, rotated rx 180 ry 0 rz 180 deg; joints [37.56, 59.213, 24.138, -142.253, 84.734, -184.064]
  Call Extruder(5332.277)
  MoveL 444 to (-54.27, -6.18, 25) mm, rotated rx 180 ry 0 rz -180 deg; joints [36.644, 58.984, 24.881, -143.198, 85.081, -183.67]
  Set speed (130.0 mm/s)
  MoveL 445 to (-49.9, -9.51, 25) mm, rotated rx 180 ry 0 rz -180 deg; joints [35.741, 59.097, 24.515, -144.089, 84.819, -183.742]
  MoveL 446 to (2.97, -12.99, 25) mm, rotated rx 180 ry 0 rz 180 deg; joints [30.614, 62.615, 14.11, -148.701, 78.603, -186.851]
  Call Extruder(5336.941)
  Set speed (80.0 mm/s)
  MoveL 447 to (5.78, -12.01, 25) mm, rotated rx -180 ry 0 rz -180 deg; joints [30.526, 62.893, 13.352, -148.739, 78.181, -187.088]
  Call Extruder(5341.605)
  MoveL 448 to (8.31, -10.42, 25) mm, rotated rx 180 ry 0 rz 180 deg; joints [30.538, 63.181, 12.572, -148.672, 77.762, -187.352]
  Call Extruder(5346.269)
  MoveL 449 to (10.42, -8.31, 25) mm, rotated rx -180 ry 0 rz -180 deg; joints [30.649, 63.464, 11.811, -148.505, 77.369, -187.631]
  Call Extruder(5350.932)
  MoveL 450 to (12.01, -5.78, 25) mm, rotated rx 180 ry 0 rz 180 deg; joints [30.85, 63.729, 11.106, -148.248, 77.022, -187.912]
  Call Extruder(5355.596)
  MoveL 451 to (12.99, -2.97, 25) mm, rotated rx -180 ry 0 rz 180 deg; joints [31.131, 63.961, 10.493, -147.916, 76.738, -188.184]
  Call Extruder(5360.260)
  MoveL 452 to (13.33, 0, 25) mm, rotated rx 180 ry 0 rz -180 deg; joints [31.476, 64.148, 10.003, -147.527, 76.53, -188.432]
  Call Extruder(5364.924)
  MoveL 453 to (12.99, 2.97, 25) mm, rotated rx -180 ry 0 rz -180 deg; joints [31.869, 64.279, 9.659, -147.099, 76.41, -188.643]
  Call Extruder(5369.587)
  MoveL 454 to (12.01, 5.78, 25) mm, rotated rx 180 ry 0 rz -180 deg; joints [32.292, 64.347, 9.481, -146.655, 76.382, -188.807]
  Call Extruder(5374.251)
  MoveL 455 to (10.42, 8.31, 25) mm, rotated rx 180 ry 0 rz 180 deg; joints [32.725, 64.349, 9.475, -146.214, 76.446, -188.912]
  Call Extruder(5378.915)
  MoveL 456 to (8.31, 10.42, 25) mm, rotated rx 180 ry 0 rz -180 deg; joints [33.149, 64.285, 9.644, -145.797, 76.598, -188.952]
  Call Extruder(5383.579)
  MoveL 457 to (5.78, 12.01, 25) mm, rotated rx 180 ry 0 rz -180 deg; joints [33.544, 64.157, 9.978, -145.423, 76.83, -188.925]
  Call Extruder(5388.243)
  MoveL 458 to (2.97, 13, 25) mm, rotated rx 180 ry 0 rz -180 deg; joints [33.893, 63.973, 10.461, -145.109, 77.129, -188.83]
  Call Extruder(5392.906)
  MoveL 459 to (0, 13.33, 25) mm, rotated rx 180 ry 0 rz 180 deg; joints [34.177, 63.744, 11.067, -144.87, 77.482, -188.671]
  Call Extruder(5397.570)
  MoveL 460 to (-2.97, 13, 25) mm, rotated rx 180 ry 0 rz 180 deg; joints [34.384, 63.481, 11.768, -144.716, 77.869, -188.458]
  Call Extruder(5402.234)
  MoveL 461 to (-5.78, 12.01, 25) mm, rotated rx 180 ry 0 rz 180 deg; joints [34.5, 63.198, 12.526, -144.657, 78.275, -188.201]
  Call Extruder(5406.898)
  MoveL 462 to (-8.31, 10.42, 25) mm, rotated rx 180 ry 0 rz -180 deg; joints [34.518, 62.91, 13.306, -144.696, 78.678, -187.915]
  Call Extruder(5411.562)
  MoveL 463 to (-10.42, 8.31, 25) mm, rotated rx 180 ry 0 rz 180 deg; joints [34.436, 62.631, 14.067, -144.834, 79.061, -187.615]
  Call Extruder(5416.225)
  MoveL 464 to (-12.01, 5.78, 25) mm, rotated rx -180 ry 0 rz -180 deg; joints [34.254, 62.375, 14.772, -145.066, 79.405, -187.319]
  Call Extruder(5420.889)
  MoveL 465 to (-13, 2.97, 25) mm, rotated rx 180 ry 0 rz 180 deg; joints [33.981, 62.154, 15.385, -145.383, 79.693, -187.041]
  Call Extruder(5425.553)
  MoveL 466 to (-13.33, 0, 25) mm, rotated rx 180 ry 0 rz -180 deg; joints [33.63, 61.979, 15.875, -145.769, 79.91, -186.797]
  Call Extruder(5430.217)
  MoveL 467 to (-13, -2.97, 25) mm, rotated rx 180 ry 0 rz 180 deg; joints [33.218, 61.857, 16.218, -146.207, 80.046, -186.599]
  Call Extruder(5434.880)
  MoveL 468 to (-12.01, -5.78, 25) mm, rotated rx -180 ry 0 rz 180 deg; joints [32.767, 61.794, 16.397, -146.673, 80.091, -186.456]
  Call Extruder(5439.544)
  MoveL 469 to (-10.42, -8.31, 25) mm, rotated rx 180 ry 0 rz -180 deg; joints [32.302, 61.792, 16.402, -147.142, 80.042, -186.373]
  Call Extruder(5444.208)
  MoveL 470 to (-8.31, -10.42, 25) mm, rotated rx -180 ry 0 rz -180 deg; joints [31.85, 61.851, 16.234, -147.588, 79.9, -186.354]
  Call Extruder(5448.872)
  MoveL 471 to (-5.78, -12.01, 25) mm, rotated rx -180 ry 0 rz -180 deg; joints [31.435, 61.97, 15.9, -147.986, 79.671, -186.396]
  Call Extruder(5453.535)
  MoveL 472 to (-2.97, -12.99, 25) mm, rotated rx 180 ry 0 rz 180 deg; joints [31.079, 62.143, 15.417, -148.315, 79.368, -186.497]
  Call Extruder(5458.199)
  MoveL 473 to (0, -13.33, 25) mm, rotated rx -180 ry 0 rz -180 deg; joints [30.801, 62.361, 14.811, -148.558, 79.005, -186.651]
  Call Extruder(5462.863)
  MoveL 474 to (2.97, -12.99, 25) mm, rotated rx 180 ry 0 rz 180 deg; joints [30.614, 62.615, 14.11, -148.701, 78.603, -186.851]
  Set speed (130.0 mm/s)
  MoveL 475 to (2.97, -12.99, 30) mm, rotated rx -180 ry 0 rz 180 deg; joints [30.614, 61.666, 14.628, -148.655, 78.234, -187.08]
  MoveL 476 to (-26.25, -4.54, 30) mm, rotated rx -180 ry 0 rz 180 deg; joints [34.172, 59.845, 19.707, -145.381, 81.371, -185.913]
  Call Extruder(5465.096)
  Set speed (60.0 mm/s)
  MoveL 477 to (-26.09, -5.96, 30) mm, rotated rx -180 ry 0 rz -180 deg; joints [33.969, 59.789, 19.87, -145.595, 81.438, -185.822]
  Call Extruder(5474.461)
  MoveL 478 to (-24.12, -11.61, 30) mm, rotated rx -180 ry 0 rz -180 deg; joints [33.033, 59.664, 20.231, -146.556, 81.542, -185.549]
  Call Extruder(5483.826)
  MoveL 479 to (-20.93, -16.69, 30) mm, rotated rx -180 ry 0 rz 180 deg; joints [32.066, 59.661, 20.241, -147.531, 81.455, -185.401]
  Call Extruder(5493.191)
  MoveL 480 to (-16.69, -20.93, 30) mm, rotated rx 180 ry 0 rz -180 deg; joints [31.126, 59.778, 19.901, -148.459, 81.178, -185.378]
  Call Extruder(5502.556)
  MoveL 481 to (-11.61, -24.11, 30) mm, rotated rx 180 ry 0 rz -180 deg; joints [30.272, 60.012, 19.227, -149.284, 80.72, -185.473]
  Call Extruder(5511.921)
  MoveL 482 to (-5.96, -26.09, 30) mm, rotated rx 180 ry 0 rz -180 deg; joints [29.552, 60.353, 18.254, -149.957, 80.105, -185.676]
  Call Extruder(5521.286)
  MoveL 483 to (0, -26.77, 30) mm, rotated rx 180 ry 0 rz -180 deg; joints [29.003, 60.788, 17.033, -150.441, 79.368, -185.974]
  Call Extruder(5530.651)
  MoveL 484 to (5.96, -26.09, 30) mm, rotated rx 180 ry 0 rz 180 deg; joints [28.65, 61.299, 15.625, -150.712, 78.548, -186.355]
  Call Extruder(5540.016)
  MoveL 485 to (11.61, -24.11, 30) mm, rotated rx -180 ry 0 rz -180 deg; joints [28.503, 61.861, 14.101, -150.763, 77.692, -186.804]
  Call Extruder(5549.381)
  MoveL 486 to (16.69, -20.93, 30) mm, rotated rx 180 ry 0 rz -180 deg; joints [28.559, 62.449, 12.535, -150.597, 76.846, -187.308]
  Call Extruder(5558.746)
  MoveL 487 to (20.93, -16.69, 30) mm, rotated rx 180 ry 0 rz 180 deg; joints [28.808, 63.032, 11.007, -150.231, 76.057, -187.847]
  Call Extruder(5568.111)
  MoveL 488 to (24.12, -11.61, 30) mm, rotated rx 180 ry 0 rz 180 deg; joints [29.229, 63.581, 9.59, -149.691, 75.365, -188.402]
  Call Extruder(5577.475)
  MoveL 489 to (26.09, -5.96, 30) mm, rotated rx 180 ry 0 rz 180 deg; joints [29.796, 64.064, 8.357, -149.008, 74.806, -188.947]
  Call Extruder(5586.841)
  MoveL 490 to (26.77, 0, 30) mm, rotated rx 180 ry 0 rz 180 deg; joints [30.482, 64.455, 7.369, -148.221, 74.406, -189.455]
  Call Extruder(5596.206)
  MoveL 491 to (26.09, 5.96, 30) mm, rotated rx 180 ry 0 rz 180 deg; joints [31.252, 64.731, 6.677, -147.369, 74.183, -189.9]
  Call Extruder(5605.570)
  MoveL 492 to (24.11, 11.61, 30) mm, rotated rx -180 ry 0 rz 180 deg; joints [32.076, 64.875, 6.316, -146.493, 74.146, -190.252]
  Call Extruder(5614.935)
  MoveL 493 to (20.93, 16.69, 30) mm, rotated rx -180 ry 0 rz 180 deg; joints [32.917, 64.88, 6.306, -145.632, 74.292, -190.49]
  Call Extruder(5624.301)
  MoveL 494 to (16.69, 20.93, 30) mm, rotated rx 180 ry 0 rz -180 deg; joints [33.742, 64.743, 6.646, -144.822, 74.611, -190.595]
  Call Extruder(5633.666)
  MoveL 495 to (11.61, 24.12, 30) mm, rotated rx 180 ry 0 rz 180 deg; joints [34.517, 64.475, 7.32, -144.097, 75.083, -190.557]
  Call Extruder(5643.030)
  MoveL 496 to (5.96, 26.09, 30) mm, rotated rx 180 ry 0 rz -180 deg; joints [35.208, 64.09, 8.292, -143.485, 75.682, -190.376]
  Call Extruder(5652.395)
  MoveL 497 to (0, 26.77, 30) mm, rotated rx -180 ry 0 rz -180 deg; joints [35.784, 63.611, 9.512, -143.012, 76.378, -190.059]
  Call Extruder(5661.761)
  MoveL 498 to (-5.96, 26.09, 30) mm, rotated rx 180 ry 0 rz -180 deg; joints [36.214, 63.066, 10.92, -142.699, 77.139, -189.624]
  Call Extruder(5671.125)
  MoveL 499 to (-11.61, 24.12, 30) mm, rotated rx -180 ry 0 rz -180 deg; joints [36.473, 62.484, 12.444, -142.563, 77.93, -189.095]
  Call Extruder(5680.490)
  MoveL 500 to (-16.69, 20.93, 30) mm, rotated rx 180 ry 0 rz -180 deg; joints [36.542, 61.895, 14.009, -142.617, 78.716, -188.503]
  Call Extruder(5689.855)
  MoveL 501 to (-20.93, 16.69, 30) mm, rotated rx 180 ry 0 rz -180 deg; joints [36.407, 61.331, 15.538, -142.865, 79.464, -187.883]
  Call Extruder(5699.220)
  MoveL 502 to (-24.12, 11.61, 30) mm, rotated rx -180 ry 0 rz 180 deg; joints [36.065, 60.817, 16.955, -143.307, 80.141, -187.271]
  Call Extruder(5708.585)
  MoveL 503 to (-26.09, 5.96, 30) mm, rotated rx 180 ry 0 rz 180 deg; joints [35.528, 60.376, 18.188, -143.927, 80.715, -186.704]
  Call Extruder(5717.950)
  MoveL 504 to (-26.77, 0, 30) mm, rotated rx 180 ry 0 rz -180 deg; joints [34.817, 60.029, 19.177, -144.702, 81.156, -186.212]
  Call Extruder(5722.739)
  MoveL 505 to (-26.42, -3.05, 30) mm, rotated rx 180 ry 0 rz -180 deg; joints [34.385, 59.905, 19.534, -145.157, 81.3, -186.011]
  Set speed (130.0 mm/s)
  MoveL 506 to (-41.86, -6.29, 30) mm, rotated rx 180 ry 0 rz -180 deg; joints [35.393, 58.716, 23.056, -144.326, 83.3, -184.787]
  Call Extruder(5727.737)
  Set speed (60.0 mm/s)
  MoveL 507 to (-41.5, -9.47, 30) mm, rotated rx 180 ry 0 rz -180 deg; joints [34.924, 58.596, 23.422, -144.814, 83.463, -184.589]
  Call Extruder(5742.633)
  MoveL 508 to (-38.36, -18.47, 30) mm, rotated rx -180 ry 0 rz -180 deg; joints [33.373, 58.408, 24.003, -146.395, 83.668, -184.192]
  Call Extruder(5757.528)
  MoveL 509 to (-33.28, -26.54, 30) mm, rotated rx 180 ry 0 rz 180 deg; joints [31.763, 58.403, 24.019, -148.012, 83.562, -184.006]
  Call Extruder(5772.424)
  MoveL 510 to (-26.54, -33.28, 30) mm, rotated rx 180 ry 0 rz 180 deg; joints [30.206, 58.58, 23.472, -149.553, 83.137, -184.018]
  Call Extruder(5787.320)
  MoveL 511 to (-18.47, -38.36, 30) mm, rotated rx -180 ry 0 rz -180 deg; joints [28.808, 58.935, 22.391, -150.913, 82.406, -184.205]
  Call Extruder(5802.216)
  MoveL 512 to (-9.47, -41.5, 30) mm, rotated rx 180 ry 0 rz 180 deg; joints [27.654, 59.458, 20.834, -152.005, 81.41, -184.54]
  Call Extruder(5817.112)
  MoveL 513 to (0, -42.57, 30) mm, rotated rx -180 ry 0 rz -180 deg; joints [26.805, 60.132, 18.884, -152.767, 80.208, -185.002]
  Call Extruder(5832.007)
  MoveL 514 to (9.47, -41.5, 30) mm, rotated rx 180 ry 0 rz 180 deg; joints [26.29, 60.93, 16.64, -153.167, 78.873, -185.576]
  Call Extruder(5846.903)
  MoveL 515 to (18.47, -38.36, 30) mm, rotated rx -180 ry 0 rz 180 deg; joints [26.114, 61.819, 14.215, -153.2, 77.484, -186.247]
  Call Extruder(5861.799)
  MoveL 516 to (26.54, -33.28, 30) mm, rotated rx 180 ry 0 rz -180 deg; joints [26.262, 62.757, 11.725, -152.885, 76.118, -187.004]
  Call Extruder(5876.695)
  MoveL 517 to (33.28, -26.54, 30) mm, rotated rx 180 ry 0 rz 180 deg; joints [26.703, 63.697, 9.292, -152.254, 74.849, -187.828]
  Call Extruder(5891.591)
  MoveL 518 to (38.36, -18.47, 30) mm, rotated rx 180 ry 0 rz 180 deg; joints [27.4, 64.589, 7.033, -151.356, 73.745, -188.693]
  Call Extruder(5906.486)
  MoveL 519 to (41.5, -9.47, 30) mm, rotated rx -180 ry 0 rz 180 deg; joints [28.309, 65.381, 5.062, -150.247, 72.86, -189.563]
  Call Extruder(5921.382)
  MoveL 520 to (42.57, 0, 30) mm, rotated rx 180 ry 0 rz 180 deg; joints [29.382, 66.026, 3.478, -148.989, 72.236, -190.393]
  Call Extruder(5936.278)
  MoveL 521 to (41.5, 9.47, 30) mm, rotated rx -180 ry 0 rz -180 deg; joints [30.575, 66.484, 2.366, -147.647, 71.902, -191.133]
  Call Extruder(5951.174)
  MoveL 522 to (38.36, 18.47, 30) mm, rotated rx 180 ry 0 rz 180 deg; joints [31.839, 66.724, 1.785, -146.282, 71.867, -191.734]
  Call Extruder(5966.070)
  MoveL 523 to (33.28, 26.54, 30) mm, rotated rx -180 ry 0 rz -180 deg; joints [33.128, 66.731, 1.768, -144.955, 72.125, -192.149]
  Call Extruder(5980.965)
  MoveL 524 to (26.54, 33.29, 30) mm, rotated rx 180 ry 0 rz -180 deg; joints [34.394, 66.504, 2.316, -143.715, 72.655, -192.346]
  Call Extruder(5995.861)
  MoveL 525 to (18.47, 38.36, 30) mm, rotated rx 180 ry 0 rz 180 deg; joints [35.592, 66.059, 3.399, -142.608, 73.42, -192.304]
  Call Extruder(6010.757)
  MoveL 526 to (9.47, 41.51, 30) mm, rotated rx 180 ry 0 rz 180 deg; joints [36.675, 65.423, 4.957, -141.671, 74.377, -192.019]
  Call Extruder(6025.653)
  MoveL 527 to (0, 42.57, 30) mm, rotated rx -180 ry 0 rz 180 deg; joints [37.594, 64.639, 6.908, -140.935, 75.475, -191.507]
  Call Extruder(6040.549)
  MoveL 528 to (-9.47, 41.51, 30) mm, rotated rx 180 ry 0 rz 180 deg; joints [38.304, 63.751, 9.153, -140.43, 76.663, -190.793]
  Call Extruder(6055.444)
  MoveL 529 to (-18.47, 38.36, 30) mm, rotated rx 180 ry 0 rz 180 deg; joints [38.762, 62.813, 11.579, -140.183, 77.89, -189.921]
  Call Extruder(6070.340)
  MoveL 530 to (-26.54, 33.29, 30) mm, rotated rx 180 ry 0 rz -180 deg; joints [38.928, 61.873, 14.069, -140.217, 79.108, -188.942]
  Call Extruder(6085.236)
  MoveL 531 to (-33.29, 26.54, 30) mm, rotated rx -180 ry 0 rz 180 deg; joints [38.772, 60.98, 16.501, -140.553, 80.271, -187.916]
  Call Extruder(6100.132)
  MoveL 532 to (-38.36, 18.47, 30) mm, rotated rx 180 ry 0 rz 180 deg; joints [38.277, 60.175, 18.759, -141.199, 81.334, -186.908]
  Call Extruder(6115.027)
  MoveL 533 to (-41.51, 9.47, 30) mm, rotated rx 180 ry 0 rz 180 deg; joints [37.447, 59.494, 20.729, -142.148, 82.252, -185.981]
  Call Extruder(6129.923)
  MoveL 534 to (-42.57, 0, 30) mm, rotated rx 180 ry 0 rz -180 deg; joints [36.31, 58.961, 22.311, -143.371, 82.977, -185.194]
  Call Extruder(6137.478)
  MoveL 535 to (-42.03, -4.8, 30) mm, rotated rx 180 ry 0 rz -180 deg; joints [35.612, 58.773, 22.882, -144.099, 83.224, -184.882]
  Set speed (130.0 mm/s)
  MoveL 536 to (-54.1, -7.67, 30) mm, rotated rx 180 ry 0 rz -180 deg; joints [36.421, 57.906, 25.586, -143.402, 84.767, -183.875]
  Call Extruder(6141.550)
  Set speed (30.0 mm/s)
  MoveL 537 to (-53.59, -12.23, 30) mm, rotated rx 180 ry 0 rz 180 deg; joints [35.732, 57.742, 26.113, -144.112, 85.016, -183.597]
  Call Extruder(6152.480)
  MoveL 538 to (-49.53, -23.85, 30) mm, rotated rx 180 ry 0 rz -180 deg; joints [33.663, 57.511, 26.87, -146.21, 85.325, -183.122]
  Call Extruder(6163.411)
  MoveL 539 to (-42.98, -34.27, 30) mm, rotated rx 180 ry 0 rz -180 deg; joints [31.506, 57.504, 26.892, -148.372, 85.224, -182.935]
  Call Extruder(6174.341)
  MoveL 540 to (-34.27, -42.98, 30) mm, rotated rx -180 ry 0 rz 180 deg; joints [29.427, 57.723, 26.178, -150.434, 84.69, -183.006]
  Call Extruder(6185.271)
  MoveL 541 to (-23.85, -49.52, 30) mm, rotated rx 180 ry 0 rz -180 deg; joints [27.581, 58.163, 24.769, -152.24, 83.739, -183.285]
  Call Extruder(6196.201)
  MoveL 542 to (-12.23, -53.59, 30) mm, rotated rx -180 ry 0 rz -180 deg; joints [26.087, 58.818, 22.746, -153.666, 82.429, -183.731]
  Call Extruder(6207.131)
  MoveL 543 to (0, -54.97, 30) mm, rotated rx 180 ry 0 rz 180 deg; joints [25.019, 59.668, 20.219, -154.636, 80.845, -184.314]
  Call Extruder(6208.682)
  MoveL 544 to (1.73, -54.77, 30) mm, rotated rx -180 ry 0 rz -180 deg; joints [24.929, 59.808, 19.813, -154.708, 80.597, -184.414]
  Call Extruder(6218.062)
  MoveL 545 to (12.23, -53.59, 30) mm, rotated rx -180 ry 0 rz -180 deg; joints [24.406, 60.686, 17.317, -155.115, 79.089, -185.018]
  Call Extruder(6228.992)
  MoveL 546 to (23.85, -49.52, 30) mm, rotated rx 180 ry 0 rz 180 deg; joints [24.239, 61.83, 14.184, -155.109, 77.269, -185.838]
  Call Extruder(6239.922)
  MoveL 547 to (34.27, -42.98, 30) mm, rotated rx 180 ry 0 rz -180 deg; joints [24.487, 63.046, 10.97, -154.649, 75.487, -186.771]
  Call Extruder(6250.852)
  MoveL 548 to (42.98, -34.27, 30) mm, rotated rx 180 ry 0 rz 180 deg; joints [25.101, 64.274, 7.824, -153.789, 73.838, -187.803]
  Call Extruder(6261.782)
  MoveL 549 to (49.52, -23.85, 30) mm, rotated rx -180 ry 0 rz -180 deg; joints [26.025, 65.447, 4.899, -152.594, 72.408, -188.906]
  Call Extruder(6272.713)
  MoveL 550 to (53.59, -12.23, 30) mm, rotated rx 180 ry 0 rz 180 deg; joints [27.2, 66.495, 2.338, -151.14, 71.267, -190.037]
  Call Extruder(6283.643)
  MoveL 551 to (54.97, 0, 30) mm, rotated rx 180 ry 0 rz 180 deg; joints [28.57, 67.354, 0.274, -149.508, 70.472, -191.136]
  Call Extruder(6294.573)
  MoveL 552 to (53.59, 12.23, 30) mm, rotated rx 180 ry 0 rz 180 deg; joints [30.077, 67.966, -1.18, -147.783, 70.056, -192.131]
  Call Extruder(6305.503)
  MoveL 553 to (49.52, 23.85, 30) mm, rotated rx -180 ry 0 rz 180 deg; joints [31.665, 68.289, -1.941, -146.046, 70.034, -192.948]
  Call Extruder(6316.433)
  MoveL 554 to (42.98, 34.27, 30) mm, rotated rx 180 ry 0 rz 180 deg; joints [33.282, 68.298, -1.963, -144.371, 70.394, -193.522]
  Call Extruder(6327.364)
  MoveL 555 to (34.27, 42.98, 30) mm, rotated rx 180 ry 0 rz 180 deg; joints [34.874, 67.993, -1.245, -142.818, 71.103, -193.802]
  Call Extruder(6338.294)
  MoveL 556 to (23.85, 49.53, 30) mm, rotated rx -180 ry 0 rz -180 deg; joints [36.387, 67.398, 0.17, -141.437, 72.11, -193.761]
  Call Extruder(6349.224)
  MoveL 557 to (12.23, 53.59, 30) mm, rotated rx 180 ry 0 rz -180 deg; joints [37.766, 66.552, 2.201, -140.266, 73.353, -193.394]
  Call Extruder(6360.154)
  MoveL 558 to (0, 54.97, 30) mm, rotated rx 180 ry 0 rz 180 deg; joints [38.954, 65.513, 4.737, -139.337, 74.765, -192.72]
  Call Extruder(6371.084)
  MoveL 559 to (-12.23, 53.59, 30) mm, rotated rx -180 ry 0 rz 180 deg; joints [39.895, 64.346, 7.645, -138.683, 76.278, -191.778]
  Call Extruder(6382.015)
  MoveL 560 to (-23.85, 49.53, 30) mm, rotated rx 180 ry 0 rz -180 deg; joints [40.528, 63.119, 10.781, -138.336, 77.832, -190.623]
  Call Extruder(6392.945)
  MoveL 561 to (-34.27, 42.98, 30) mm, rotated rx 180 ry 0 rz 180 deg; joints [40.799, 61.9, 13.996, -138.332, 79.37, -189.323]
  Call Extruder(6403.875)
  MoveL 562 to (-42.98, 34.27, 30) mm, rotated rx 180 ry 0 rz 180 deg; joints [40.659, 60.751, 17.138, -138.703, 80.842, -187.959]
  Call Extruder(6414.805)
  MoveL 563 to (-49.53, 23.85, 30) mm, rotated rx -180 ry 0 rz 180 deg; joints [40.072, 59.724, 20.057, -139.476, 82.198, -186.619]
  Call Extruder(6425.735)
  MoveL 564 to (-53.59, 12.23, 30) mm, rotated rx 180 ry 0 rz -180 deg; joints [39.031, 58.862, 22.61, -140.657, 83.386, -185.394]
  Call Extruder(6436.666)
  MoveL 565 to (-54.97, 0, 30) mm, rotated rx -180 ry 0 rz -180 deg; joints [37.56, 58.196, 24.666, -142.224, 84.347, -184.366]
  Call Extruder(6442.191)
  MoveL 566 to (-54.27, -6.18, 30) mm, rotated rx 180 ry 0 rz -180 deg; joints [36.644, 57.961, 25.41, -143.171, 84.686, -183.968]
  Set speed (130.0 mm/s)
  MoveL 567 to (-49.9, -9.51, 30) mm, rotated rx -180 ry 0 rz 180 deg; joints [35.741, 58.076, 25.044, -144.062, 84.42, -184.032]
  MoveL 568 to (2.97, -12.99, 30) mm, rotated rx -180 ry 0 rz 180 deg; joints [30.614, 61.666, 14.628, -148.655, 78.234, -187.08]
  Call Extruder(6446.855)
  Set speed (80.0 mm/s)
  MoveL 569 to (5.78, -12.01, 30) mm, rotated rx -180 ry 0 rz -180 deg; joints [30.526, 61.948, 13.869, -148.692, 77.815, -187.315]
  Call Extruder(6451.518)
  MoveL 570 to (8.31, -10.42, 30) mm, rotated rx 180 ry 0 rz 180 deg; joints [30.538, 62.24, 13.089, -148.624, 77.4, -187.577]
  Call Extruder(6456.183)
  MoveL 571 to (10.42, -8.31, 30) mm, rotated rx 180 ry 0 rz 180 deg; joints [30.649, 62.527, 12.329, -148.455, 77.012, -187.856]
  Call Extruder(6460.846)
  MoveL 572 to (12.01, -5.78, 30) mm, rotated rx 180 ry 0 rz 180 deg; joints [30.85, 62.796, 11.624, -148.197, 76.668, -188.137]
  Call Extruder(6465.510)
  MoveL 573 to (12.99, -2.97, 30) mm, rotated rx -180 ry 0 rz 180 deg; joints [31.131, 63.031, 11.011, -147.864, 76.388, -188.41]
  Call Extruder(6470.174)
  MoveL 574 to (13.33, 0, 30) mm, rotated rx -180 ry 0 rz 180 deg; joints [31.476, 63.22, 10.521, -147.473, 76.185, -188.659]
  Call Extruder(6474.838)
  MoveL 575 to (12.99, 2.97, 30) mm, rotated rx 180 ry 0 rz -180 deg; joints [31.869, 63.352, 10.177, -147.045, 76.067, -188.872]
  Call Extruder(6479.501)
  MoveL 576 to (12.01, 5.78, 30) mm, rotated rx 180 ry 0 rz 180 deg; joints [32.292, 63.422, 9.999, -146.6, 76.042, -189.037]
  Call Extruder(6484.165)
  MoveL 577 to (10.42, 8.31, 30) mm, rotated rx 180 ry 0 rz 180 deg; joints [32.725, 63.424, 9.993, -146.158, 76.108, -189.145]
  Call Extruder(6488.829)
  MoveL 578 to (8.31, 10.42, 30) mm, rotated rx 180 ry 0 rz 180 deg; joints [33.149, 63.358, 10.162, -145.742, 76.261, -189.189]
  Call Extruder(6493.493)
  MoveL 579 to (5.78, 12.01, 30) mm, rotated rx -180 ry 0 rz -180 deg; joints [33.544, 63.229, 10.496, -145.368, 76.493, -189.164]
  Call Extruder(6498.156)
  MoveL 580 to (2.97, 12.99, 30) mm, rotated rx -180 ry 0 rz 180 deg; joints [33.893, 63.043, 10.978, -145.055, 76.791, -189.072]
  Call Extruder(6502.820)
  MoveL 581 to (0, 13.33, 30) mm, rotated rx 180 ry 0 rz 180 deg; joints [34.177, 62.811, 11.585, -144.816, 77.142, -188.917]
  Call Extruder(6507.484)
  MoveL 582 to (-2.97, 12.99, 30) mm, rotated rx 180 ry 0 rz 180 deg; joints [34.384, 62.544, 12.285, -144.663, 77.527, -188.706]
  Call Extruder(6512.148)
  MoveL 583 to (-5.78, 12.01, 30) mm, rotated rx 180 ry 0 rz 180 deg; joints [34.5, 62.257, 13.044, -144.605, 77.929, -188.452]
  Call Extruder(6516.811)
  MoveL 584 to (-8.31, 10.42, 30) mm, rotated rx -180 ry 0 rz -180 deg; joints [34.518, 61.965, 13.823, -144.646, 78.329, -188.167]
  Call Extruder(6521.476)
  MoveL 585 to (-10.42, 8.31, 30) mm, rotated rx -180 ry 0 rz -180 deg; joints [34.436, 61.682, 14.584, -144.785, 78.708, -187.869]
  Call Extruder(6526.139)
  MoveL 586 to (-12.01, 5.78, 30) mm, rotated rx 180 ry 0 rz 180 deg; joints [34.254, 61.422, 15.289, -145.019, 79.048, -187.573]
  Call Extruder(6530.803)
  MoveL 587 to (-13, 2.97, 30) mm, rotated rx -180 ry 0 rz 180 deg; joints [33.981, 61.197, 15.903, -145.336, 79.332, -187.295]
  Call Extruder(6535.467)
  MoveL 588 to (-13.33, 0, 30) mm, rotated rx -180 ry 0 rz -180 deg; joints [33.63, 61.019, 16.393, -145.724, 79.545, -187.05]
  Call Extruder(6540.131)
  MoveL 589 to (-13, -2.97, 30) mm, rotated rx 180 ry 0 rz 180 deg; joints [33.218, 60.895, 16.737, -146.163, 79.677, -186.85]
  Call Extruder(6544.794)
  MoveL 590 to (-12.01, -5.78, 30) mm, rotated rx 180 ry 0 rz -180 deg; joints [32.767, 60.831, 16.915, -146.629, 79.719, -186.704]
  Call Extruder(6549.458)
  MoveL 591 to (-10.42, -8.31, 30) mm, rotated rx -180 ry 0 rz -180 deg; joints [32.302, 60.829, 16.921, -147.099, 79.668, -186.619]
  Call Extruder(6554.122)
  MoveL 592 to (-8.31, -10.42, 30) mm, rotated rx 180 ry 0 rz -180 deg; joints [31.85, 60.89, 16.752, -147.544, 79.525, -186.595]
  Call Extruder(6558.786)
  MoveL 593 to (-5.78, -12.01, 30) mm, rotated rx 180 ry 0 rz -180 deg; joints [31.435, 61.01, 16.418, -147.943, 79.297, -186.634]
  Call Extruder(6563.449)
  MoveL 594 to (-2.97, -12.99, 30) mm, rotated rx 180 ry 0 rz -180 deg; joints [31.079, 61.186, 15.935, -148.271, 78.995, -186.732]
  Call Extruder(6568.113)
  MoveL 595 to (0, -13.33, 30) mm, rotated rx 180 ry 0 rz 180 deg; joints [30.801, 61.407, 15.328, -148.513, 78.634, -186.883]
  Call Extruder(6572.777)
  MoveL 596 to (2.97, -12.99, 30) mm, rotated rx -180 ry 0 rz 180 deg; joints [30.614, 61.666, 14.628, -148.655, 78.234, -187.08]
  Set speed (130.0 mm/s)
  MoveL 597 to (2.97, -12.99, 35) mm, rotated rx 180 ry 0 rz 180 deg; joints [30.614, 60.72, 15.128, -148.606, 77.853, -187.317]
  MoveL 598 to (-26.25, -4.54, 35) mm, rotated rx 180 ry 0 rz 180 deg; joints [34.172, 58.867, 20.211, -145.339, 80.981, -186.186]
  Call Extruder(6575.010)
  Set speed (60.0 mm/s)
  MoveL 599 to (-26.09, -5.96, 35) mm, rotated rx 180 ry 0 rz 180 deg; joints [33.969, 58.809, 20.374, -145.553, 81.046, -186.094]
  Call Extruder(6584.375)
  MoveL 600 to (-24.12, -11.61, 35) mm, rotated rx -180 ry 0 rz -180 deg; joints [33.033, 58.682, 20.736, -146.516, 81.143, -185.815]
  Call Extruder(6593.739)
  MoveL 601 to (-20.93, -16.69, 35) mm, rotated rx 180 ry 0 rz -180 deg; joints [32.066, 58.679, 20.746, -147.491, 81.052, -185.661]
  Call Extruder(6603.105)
  MoveL 602 to (-16.69, -20.93, 35) mm, rotated rx -180 ry 0 rz 180 deg; joints [31.126, 58.798, 20.405, -148.419, 80.772, -185.63]
  Call Extruder(6612.470)
  MoveL 603 to (-11.61, -24.11, 35) mm, rotated rx 180 ry 0 rz -180 deg; joints [30.272, 59.037, 19.73, -149.243, 80.314, -185.717]
  Call Extruder(6621.834)
  MoveL 604 to (-5.96, -26.09, 35) mm, rotated rx 180 ry 0 rz -180 deg; joints [29.552, 59.385, 18.757, -149.915, 79.702, -185.913]
  Call Extruder(6631.200)
  MoveL 605 to (0, -26.77, 35) mm, rotated rx 180 ry 0 rz 180 deg; joints [29.003, 59.828, 17.535, -150.397, 78.969, -186.204]
  Call Extruder(6640.565)
  MoveL 606 to (5.96, -26.09, 35) mm, rotated rx 180 ry 0 rz -180 deg; joints [28.65, 60.347, 16.126, -150.667, 78.155, -186.58]
  Call Extruder(6649.929)
  MoveL 607 to (11.61, -24.11, 35) mm, rotated rx 180 ry 0 rz -180 deg; joints [28.503, 60.918, 14.601, -150.715, 77.306, -187.026]
  Call Extruder(6659.294)
  MoveL 608 to (16.69, -20.93, 35) mm, rotated rx 180 ry 0 rz -180 deg; joints [28.559, 61.515, 13.036, -150.546, 76.468, -187.527]
  Call Extruder(6668.660)
  MoveL 609 to (20.93, -16.69, 35) mm, rotated rx 180 ry 0 rz -180 deg; joints [28.808, 62.106, 11.507, -150.178, 75.688, -188.065]
  Call Extruder(6678.024)
  MoveL 610 to (24.12, -11.61, 35) mm, rotated rx 180 ry 0 rz -180 deg; joints [29.229, 62.661, 10.091, -149.635, 75.004, -188.62]
  Call Extruder(6687.389)
  MoveL 611 to (26.09, -5.96, 35) mm, rotated rx 180 ry 0 rz 180 deg; joints [29.796, 63.15, 8.859, -148.95, 74.453, -189.167]
  Call Extruder(6696.754)
  MoveL 612 to (26.77, 0, 35) mm, rotated rx 180 ry 0 rz -180 deg; joints [30.482, 63.546, 7.872, -148.16, 74.06, -189.678]
  Call Extruder(6706.119)
  MoveL 613 to (26.09, 5.96, 35) mm, rotated rx -180 ry 0 rz -180 deg; joints [31.252, 63.824, 7.18, -147.307, 73.844, -190.126]
  Call Extruder(6715.484)
  MoveL 614 to (24.11, 11.61, 35) mm, rotated rx -180 ry 0 rz -180 deg; joints [32.076, 63.97, 6.82, -146.429, 73.811, -190.483]
  Call Extruder(6724.849)
  MoveL 615 to (20.93, 16.69, 35) mm, rotated rx 180 ry 0 rz 180 deg; joints [32.917, 63.975, 6.809, -145.567, 73.961, -190.725]
  Call Extruder(6734.214)
  MoveL 616 to (16.69, 20.93, 35) mm, rotated rx -180 ry 0 rz -180 deg; joints [33.742, 63.837, 7.149, -144.757, 74.281, -190.836]
  Call Extruder(6743.579)
  MoveL 617 to (11.61, 24.12, 35) mm, rotated rx 180 ry 0 rz 180 deg; joints [34.517, 63.565, 7.822, -144.032, 74.753, -190.804]
  Call Extruder(6752.944)
  MoveL 618 to (5.96, 26.09, 35) mm, rotated rx 180 ry 0 rz -180 deg; joints [35.208, 63.176, 8.793, -143.421, 75.351, -190.629]
  Call Extruder(6762.309)
  MoveL 619 to (0, 26.77, 35) mm, rotated rx 180 ry 0 rz 180 deg; joints [35.784, 62.692, 10.013, -142.95, 76.044, -190.319]
  Call Extruder(6771.674)
  MoveL 620 to (-5.96, 26.09, 35) mm, rotated rx 180 ry 0 rz 180 deg; joints [36.214, 62.14, 11.42, -142.639, 76.801, -189.889]
  Call Extruder(6781.039)
  MoveL 621 to (-11.61, 24.12, 35) mm, rotated rx 180 ry 0 rz -180 deg; joints [36.473, 61.55, 12.944, -142.506, 77.586, -189.365]
  Call Extruder(6790.404)
  MoveL 622 to (-16.69, 20.93, 35) mm, rotated rx 180 ry 0 rz -180 deg; joints [36.542, 60.953, 14.509, -142.562, 78.365, -188.777]
  Call Extruder(6799.769)
  MoveL 623 to (-20.93, 16.69, 35) mm, rotated rx -180 ry 0 rz 180 deg; joints [36.407, 60.379, 16.039, -142.814, 79.105, -188.16]
  Call Extruder(6809.134)
  MoveL 624 to (-24.12, 11.61, 35) mm, rotated rx -180 ry 0 rz -180 deg; joints [36.065, 59.856, 17.456, -143.258, 79.774, -187.55]
  Call Extruder(6818.499)
  MoveL 625 to (-26.09, 5.96, 35) mm, rotated rx 180 ry 0 rz -180 deg; joints [35.528, 59.408, 18.691, -143.881, 80.339, -186.982]
  Call Extruder(6827.864)
  MoveL 626 to (-26.77, 0, 35) mm, rotated rx -180 ry 0 rz 180 deg; joints [34.817, 59.054, 19.681, -144.659, 80.771, -186.488]
  Call Extruder(6832.653)
  MoveL 627 to (-26.42, -3.05, 35) mm, rotated rx -180 ry 0 rz -180 deg; joints [34.385, 58.928, 20.038, -145.115, 80.912, -186.284]
  Set speed (130.0 mm/s)
  MoveL 628 to (-41.86, -6.29, 35) mm, rotated rx 180 ry 0 rz -180 deg; joints [35.393, 57.713, 23.565, -144.292, 82.899, -185.078]
  Call Extruder(6837.651)
  Set speed (60.0 mm/s)
  MoveL 629 to (-41.51, -9.47, 35) mm, rotated rx 180 ry 0 rz 180 deg; joints [34.924, 57.59, 23.931, -144.78, 83.057, -184.878]
  Call Extruder(6852.546)
  MoveL 630 to (-38.36, -18.47, 35) mm, rotated rx -180 ry 0 rz -180 deg; joints [33.373, 57.398, 24.513, -146.363, 83.251, -184.471]
  Call Extruder(6867.442)
